      "I830.5" { ExternalVisible := 'False'} : Bool := FALSE;   // I830.5
      "I830.6" { ExternalVisible := 'False'} : Bool := FALSE;   // I830.6
      "I830.7" { ExternalVisible := 'False'} : Bool := FALSE;   // I830.7
      "I831.0" { ExternalVisible := 'False'} : Bool := FALSE;   // I831.0
      "I831.1" { ExternalVisible := 'False'} : Bool := FALSE;   // I831.1
      "I831.2" { ExternalVisible := 'False'} : Bool := FALSE;   // I831.2
      "I831.3" { ExternalVisible := 'False'} : Bool := FALSE;   // I831.3
      "I831.4" { ExternalVisible := 'False'} : Bool := FALSE;   // I831.4
      "I831.5" { ExternalVisible := 'False'} : Bool := FALSE;   // I831.5
      "I831.6" { ExternalVisible := 'False'} : Bool := FALSE;   // I831.6
      "I831.7" { ExternalVisible := 'False'} : Bool := FALSE;   // I831.7
      "I832.0" { ExternalVisible := 'False'} : Bool := FALSE;   // I832.0
      "I832.1" { ExternalVisible := 'False'} : Bool := FALSE;   // I832.1
      "I832.2" { ExternalVisible := 'False'} : Bool := FALSE;   // I832.2
      "I832.3" { ExternalVisible := 'False'} : Bool := FALSE;   // I832.3
      "I832.4" { ExternalVisible := 'False'} : Bool := FALSE;   // I832.4
      "I832.5" { ExternalVisible := 'False'} : Bool := FALSE;   // I832.5
      "I832.6" { ExternalVisible := 'False'} : Bool := FALSE;   // I832.6
      "I832.7" { ExternalVisible := 'False'} : Bool := FALSE;   // I832.7
      "I833.0" { ExternalVisible := 'False'} : Bool := FALSE;   // I833.0
      "I833.1" { ExternalVisible := 'False'} : Bool := FALSE;   // I833.1
      "I833.2" { ExternalVisible := 'False'} : Bool := FALSE;   // I833.2
      "I833.3" { ExternalVisible := 'False'} : Bool := FALSE;   // I833.3
      "I833.4" { ExternalVisible := 'False'} : Bool := FALSE;   // I833.4
      "I833.5" { ExternalVisible := 'False'} : Bool := FALSE;   // I833.5
      "I833.6" { ExternalVisible := 'False'} : Bool := FALSE;   // I833.6
      "I833.7" { ExternalVisible := 'False'} : Bool := FALSE;   // I833.7
      "I834.0" { ExternalVisible := 'False'} : Bool := FALSE;   // I834.0
      "I834.1" { ExternalVisible := 'False'} : Bool := FALSE;   // I834.1
      "I834.2" { ExternalVisible := 'False'} : Bool := FALSE;   // I834.2
      "I834.3" { ExternalVisible := 'False'} : Bool := FALSE;   // I834.3
      "I834.4" { ExternalVisible := 'False'} : Bool := FALSE;   // I834.4
      "I834.5" { ExternalVisible := 'False'} : Bool := FALSE;   // I834.5
      "I834.6" { ExternalVisible := 'False'} : Bool := FALSE;   // I834.6
      "I834.7" { ExternalVisible := 'False'} : Bool := FALSE;   // I834.7
      "I835.0" { ExternalVisible := 'False'} : Bool := FALSE;   // I835.0
      "I835.1" { ExternalVisible := 'False'} : Bool := FALSE;   // I835.1
      "I835.2" { ExternalVisible := 'False'} : Bool := FALSE;   // I835.2
      "I835.3" { ExternalVisible := 'False'} : Bool := FALSE;   // I835.3
      "I835.4" { ExternalVisible := 'False'} : Bool := FALSE;   // I835.4
      "I835.5" { ExternalVisible := 'False'} : Bool := FALSE;   // I835.5
      "I835.6" { ExternalVisible := 'False'} : Bool := FALSE;   // I835.6
      "I835.7" { ExternalVisible := 'False'} : Bool := FALSE;   // I835.7
      "I836.0" { ExternalVisible := 'False'} : Bool := FALSE;   // I836.0
      "I836.1" { ExternalVisible := 'False'} : Bool := FALSE;   // I836.1
      "I836.2" { ExternalVisible := 'False'} : Bool := FALSE;   // I836.2
      "I836.3" { ExternalVisible := 'False'} : Bool := FALSE;   // I836.3
      "I836.4" { ExternalVisible := 'False'} : Bool := FALSE;   // I836.4
      "I836.5" { ExternalVisible := 'False'} : Bool := FALSE;   // I836.5
      "I836.6" { ExternalVisible := 'False'} : Bool := FALSE;   // I836.6
      "I836.7" { ExternalVisible := 'False'} : Bool := FALSE;   // I836.7
      "I837.0" { ExternalVisible := 'False'} : Bool := FALSE;   // I837.0
      "I837.1" { ExternalVisible := 'False'} : Bool := FALSE;   // I837.1
      "I837.2" { ExternalVisible := 'False'} : Bool := FALSE;   // I837.2
      "I837.3" { ExternalVisible := 'False'} : Bool := FALSE;   // I837.3
      "I837.4" { ExternalVisible := 'False'} : Bool := FALSE;   // I837.4
      "I837.5" { ExternalVisible := 'False'} : Bool := FALSE;   // I837.5
      "I837.6" { ExternalVisible := 'False'} : Bool := FALSE;   // I837.6
      "I837.7" { ExternalVisible := 'False'} : Bool := FALSE;   // I837.7
      "I838.0" { ExternalVisible := 'False'} : Bool := FALSE;   // I838.0
      "I838.1" { ExternalVisible := 'False'} : Bool := FALSE;   // I838.1
      "I838.2" { ExternalVisible := 'False'} : Bool := FALSE;   // I838.2
      "I838.3" { ExternalVisible := 'False'} : Bool := FALSE;   // I838.3
      "I838.4" { ExternalVisible := 'False'} : Bool := FALSE;   // I838.4
      "I838.5" { ExternalVisible := 'False'} : Bool := FALSE;   // I838.5
      "I838.6" { ExternalVisible := 'False'} : Bool := FALSE;   // I838.6
      "I838.7" { ExternalVisible := 'False'} : Bool := FALSE;   // I838.7
      "I839.0" { ExternalVisible := 'False'} : Bool := FALSE;   // I839.0
      "I839.1" { ExternalVisible := 'False'} : Bool := FALSE;   // I839.1
      "I839.2" { ExternalVisible := 'False'} : Bool := FALSE;   // I839.2
      "I839.3" { ExternalVisible := 'False'} : Bool := FALSE;   // I839.3
      "I839.4" { ExternalVisible := 'False'} : Bool := FALSE;   // I839.4
      "I839.5" { ExternalVisible := 'False'} : Bool := FALSE;   // I839.5
      "I839.6" { ExternalVisible := 'False'} : Bool := FALSE;   // I839.6
      "I839.7" { ExternalVisible := 'False'} : Bool := FALSE;   // I839.7
      "I840.0" { ExternalVisible := 'False'} : Bool := FALSE;   // I840.0
      "I840.1" { ExternalVisible := 'False'} : Bool := FALSE;   // I840.1
      "I840.2" { ExternalVisible := 'False'} : Bool := FALSE;   // I840.2
      "I840.3" { ExternalVisible := 'False'} : Bool := FALSE;   // I840.3
      "I840.4" { ExternalVisible := 'False'} : Bool := FALSE;   // I840.4
      "I840.5" { ExternalVisible := 'False'} : Bool := FALSE;   // I840.5
      "I840.6" { ExternalVisible := 'False'} : Bool := FALSE;   // I840.6
      "I840.7" { ExternalVisible := 'False'} : Bool := FALSE;   // I840.7
      "I841.0" { ExternalVisible := 'False'} : Bool := FALSE;   // I841.0
      "I841.1" { ExternalVisible := 'False'} : Bool := FALSE;   // I841.1
      "I841.2" { ExternalVisible := 'False'} : Bool := FALSE;   // I841.2
      "I841.3" { ExternalVisible := 'False'} : Bool := FALSE;   // I841.3
      "I841.4" { ExternalVisible := 'False'} : Bool := FALSE;   // I841.4
      "I841.5" { ExternalVisible := 'False'} : Bool := FALSE;   // I841.5
      "I841.6" { ExternalVisible := 'False'} : Bool := FALSE;   // I841.6
      "I841.7" { ExternalVisible := 'False'} : Bool := FALSE;   // I841.7
      "I842.0" { ExternalVisible := 'False'} : Bool := FALSE;   // I842.0
      "I842.1" { ExternalVisible := 'False'} : Bool := FALSE;   // I842.1
      "I842.2" { ExternalVisible := 'False'} : Bool := FALSE;   // I842.2
      "I842.3" { ExternalVisible := 'False'} : Bool := FALSE;   // I842.3
      "I842.4" { ExternalVisible := 'False'} : Bool := FALSE;   // I842.4
      "I842.5" { ExternalVisible := 'False'} : Bool := FALSE;   // I842.5
      "I842.6" { ExternalVisible := 'False'} : Bool := FALSE;   // I842.6
      "I842.7" { ExternalVisible := 'False'} : Bool := FALSE;   // I842.7
      "I843.0" { ExternalVisible := 'False'} : Bool := FALSE;   // I843.0
      "I843.1" { ExternalVisible := 'False'} : Bool := FALSE;   // I843.1
      "I843.2" { ExternalVisible := 'False'} : Bool := FALSE;   // I843.2
      "I843.3" { ExternalVisible := 'False'} : Bool := FALSE;   // I843.3
      "I843.4" { ExternalVisible := 'False'} : Bool := FALSE;   // I843.4
      "I843.5" { ExternalVisible := 'False'} : Bool := FALSE;   // I843.5
      "I843.6" { ExternalVisible := 'False'} : Bool := FALSE;   // I843.6
      "I843.7" { ExternalVisible := 'False'} : Bool := FALSE;   // I843.7
      "I844.0" { ExternalVisible := 'False'} : Bool := FALSE;   // I844.0
      "I844.1" { ExternalVisible := 'False'} : Bool := FALSE;   // I844.1
      "I844.2" { ExternalVisible := 'False'} : Bool := FALSE;   // I844.2
      "I844.3" { ExternalVisible := 'False'} : Bool := FALSE;   // I844.3
      "I844.4" { ExternalVisible := 'False'} : Bool := FALSE;   // I844.4
      "I844.5" { ExternalVisible := 'False'} : Bool := FALSE;   // I844.5
      "I844.6" { ExternalVisible := 'False'} : Bool := FALSE;   // I844.6
      "I844.7" { ExternalVisible := 'False'} : Bool := FALSE;   // I844.7
      "I845.0" { ExternalVisible := 'False'} : Bool := FALSE;   // I845.0
      "I845.1" { ExternalVisible := 'False'} : Bool := FALSE;   // I845.1
      "I845.2" { ExternalVisible := 'False'} : Bool := FALSE;   // I845.2
      "I845.3" { ExternalVisible := 'False'} : Bool := FALSE;   // I845.3
      "I845.4" { ExternalVisible := 'False'} : Bool := FALSE;   // I845.4
      "I845.5" { ExternalVisible := 'False'} : Bool := FALSE;   // I845.5
      "I845.6" { ExternalVisible := 'False'} : Bool := FALSE;   // I845.6
      "I845.7" { ExternalVisible := 'False'} : Bool := FALSE;   // I845.7
      "I846.0" { ExternalVisible := 'False'} : Bool := FALSE;   // I846.0
      "I846.1" { ExternalVisible := 'False'} : Bool := FALSE;   // I846.1
      "I846.2" { ExternalVisible := 'False'} : Bool := FALSE;   // I846.2
      "I846.3" { ExternalVisible := 'False'} : Bool := FALSE;   // I846.3
      "I846.4" { ExternalVisible := 'False'} : Bool := FALSE;   // I846.4
      "I846.5" { ExternalVisible := 'False'} : Bool := FALSE;   // I846.5
      "I846.6" { ExternalVisible := 'False'} : Bool := FALSE;   // I846.6
      "I846.7" { ExternalVisible := 'False'} : Bool := FALSE;   // I846.7
      "I847.0" { ExternalVisible := 'False'} : Bool := FALSE;   // I847.0
      "I847.1" { ExternalVisible := 'False'} : Bool := FALSE;   // I847.1
      "I847.2" { ExternalVisible := 'False'} : Bool := FALSE;   // I847.2
      "I847.3" { ExternalVisible := 'False'} : Bool := FALSE;   // I847.3
      "I847.4" { ExternalVisible := 'False'} : Bool := FALSE;   // I847.4
      "I847.5" { ExternalVisible := 'False'} : Bool := FALSE;   // I847.5
      "I847.6" { ExternalVisible := 'False'} : Bool := FALSE;   // I847.6
      "I847.7" { ExternalVisible := 'False'} : Bool := FALSE;   // I847.7
      "I848.0" { ExternalVisible := 'False'} : Bool := FALSE;   // I848.0
      "I848.1" { ExternalVisible := 'False'} : Bool := FALSE;   // I848.1
      "I848.2" { ExternalVisible := 'False'} : Bool := FALSE;   // I848.2
      "I848.3" { ExternalVisible := 'False'} : Bool := FALSE;   // I848.3
      "I848.4" { ExternalVisible := 'False'} : Bool := FALSE;   // I848.4
      "I848.5" { ExternalVisible := 'False'} : Bool := FALSE;   // I848.5
      "I848.6" { ExternalVisible := 'False'} : Bool := FALSE;   // I848.6
      "I848.7" { ExternalVisible := 'False'} : Bool := FALSE;   // I848.7
      "I849.0" { ExternalVisible := 'False'} : Bool := FALSE;   // I849.0
      "I849.1" { ExternalVisible := 'False'} : Bool := FALSE;   // I849.1
      "I849.2" { ExternalVisible := 'False'} : Bool := FALSE;   // I849.2
      "I849.3" { ExternalVisible := 'False'} : Bool := FALSE;   // I849.3
      "I849.4" { ExternalVisible := 'False'} : Bool := FALSE;   // I849.4
      "I849.5" { ExternalVisible := 'False'} : Bool := FALSE;   // I849.5
      "I849.6" { ExternalVisible := 'False'} : Bool := FALSE;   // I849.6
      "I849.7" { ExternalVisible := 'False'} : Bool := FALSE;   // I849.7
      "I850.0" { ExternalVisible := 'False'} : Bool := FALSE;   // I850.0
      "I850.1" { ExternalVisible := 'False'} : Bool := FALSE;   // I850.1
      "I850.2" { ExternalVisible := 'False'} : Bool := FALSE;   // I850.2
      "I850.3" { ExternalVisible := 'False'} : Bool := FALSE;   // I850.3
      "I850.4" { ExternalVisible := 'False'} : Bool := FALSE;   // I850.4
      "I850.5" { ExternalVisible := 'False'} : Bool := FALSE;   // I850.5
      "I850.6" { ExternalVisible := 'False'} : Bool := FALSE;   // I850.6
      "I850.7" { ExternalVisible := 'False'} : Bool := FALSE;   // I850.7
      "I851.0" { ExternalVisible := 'False'} : Bool := FALSE;   // I851.0
      "I851.1" { ExternalVisible := 'False'} : Bool := FALSE;   // I851.1
      "I851.2" { ExternalVisible := 'False'} : Bool := FALSE;   // I851.2
      "I851.3" { ExternalVisible := 'False'} : Bool := FALSE;   // I851.3
      "I851.4" { ExternalVisible := 'False'} : Bool := FALSE;   // I851.4
      "I851.5" { ExternalVisible := 'False'} : Bool := FALSE;   // I851.5
      "I851.6" { ExternalVisible := 'False'} : Bool := FALSE;   // I851.6
      "I851.7" { ExternalVisible := 'False'} : Bool := FALSE;   // I851.7
      "I852.0" { ExternalVisible := 'False'} : Bool := FALSE;   // I852.0
      "I852.1" { ExternalVisible := 'False'} : Bool := FALSE;   // I852.1
      "I852.2" { ExternalVisible := 'False'} : Bool := FALSE;   // I852.2
      "I852.3" { ExternalVisible := 'False'} : Bool := FALSE;   // I852.3
      "I852.4" { ExternalVisible := 'False'} : Bool := FALSE;   // I852.4
      "I852.5" { ExternalVisible := 'False'} : Bool := FALSE;   // I852.5
      "I852.6" { ExternalVisible := 'False'} : Bool := FALSE;   // I852.6
      "I852.7" { ExternalVisible := 'False'} : Bool := FALSE;   // I852.7
      "I853.0" { ExternalVisible := 'False'} : Bool := FALSE;   // I853.0
      "I853.1" { ExternalVisible := 'False'} : Bool := FALSE;   // I853.1
      "I853.2" { ExternalVisible := 'False'} : Bool := FALSE;   // I853.2
      "I853.3" { ExternalVisible := 'False'} : Bool := FALSE;   // I853.3
      "I853.4" { ExternalVisible := 'False'} : Bool := FALSE;   // I853.4
      "I853.5" { ExternalVisible := 'False'} : Bool := FALSE;   // I853.5
      "I853.6" { ExternalVisible := 'False'} : Bool := FALSE;   // I853.6
      "I853.7" { ExternalVisible := 'False'} : Bool := FALSE;   // I853.7
      "I854.0" { ExternalVisible := 'False'} : Bool := FALSE;   // I854.0
      "I854.1" { ExternalVisible := 'False'} : Bool := FALSE;   // I854.1
      "I854.2" { ExternalVisible := 'False'} : Bool := FALSE;   // I854.2
      "I854.3" { ExternalVisible := 'False'} : Bool := FALSE;   // I854.3
      "I854.4" { ExternalVisible := 'False'} : Bool := FALSE;   // I854.4
      "I854.5" { ExternalVisible := 'False'} : Bool := FALSE;   // I854.5
      "I854.6" { ExternalVisible := 'False'} : Bool := FALSE;   // I854.6
      "I854.7" { ExternalVisible := 'False'} : Bool := FALSE;   // I854.7
      "I855.0" { ExternalVisible := 'False'} : Bool := FALSE;   // I855.0
      "I855.1" { ExternalVisible := 'False'} : Bool := FALSE;   // I855.1
      "I855.2" { ExternalVisible := 'False'} : Bool := FALSE;   // I855.2
      "I855.3" { ExternalVisible := 'False'} : Bool := FALSE;   // I855.3
      "I855.4" { ExternalVisible := 'False'} : Bool := FALSE;   // I855.4
      "I855.5" { ExternalVisible := 'False'} : Bool := FALSE;   // I855.5
      "I855.6" { ExternalVisible := 'False'} : Bool := FALSE;   // I855.6
      "I855.7" { ExternalVisible := 'False'} : Bool := FALSE;   // I855.7
      "I856.0" { ExternalVisible := 'False'} : Bool := FALSE;   // I856.0
      "I856.1" { ExternalVisible := 'False'} : Bool := FALSE;   // I856.1
      "I856.2" { ExternalVisible := 'False'} : Bool := FALSE;   // I856.2
      "I856.3" { ExternalVisible := 'False'} : Bool := FALSE;   // I856.3
      "I856.4" { ExternalVisible := 'False'} : Bool := FALSE;   // I856.4
      "I856.5" { ExternalVisible := 'False'} : Bool := FALSE;   // I856.5
      "I856.6" { ExternalVisible := 'False'} : Bool := FALSE;   // I856.6
      "I856.7" { ExternalVisible := 'False'} : Bool := FALSE;   // I856.7
      "I857.0" { ExternalVisible := 'False'} : Bool := FALSE;   // I857.0
      "I857.1" { ExternalVisible := 'False'} : Bool := FALSE;   // I857.1
      "I857.2" { ExternalVisible := 'False'} : Bool := FALSE;   // I857.2
      "I857.3" { ExternalVisible := 'False'} : Bool := FALSE;   // I857.3
      "I857.4" { ExternalVisible := 'False'} : Bool := FALSE;   // I857.4
      "I857.5" { ExternalVisible := 'False'} : Bool := FALSE;   // I857.5
      "I857.6" { ExternalVisible := 'False'} : Bool := FALSE;   // I857.6
      "I857.7" { ExternalVisible := 'False'} : Bool := FALSE;   // I857.7
      "I858.0" { ExternalVisible := 'False'} : Bool := FALSE;   // I858.0
      "I858.1" { ExternalVisible := 'False'} : Bool := FALSE;   // I858.1
      "I858.2" { ExternalVisible := 'False'} : Bool := FALSE;   // I858.2
      "I858.3" { ExternalVisible := 'False'} : Bool := FALSE;   // I858.3
      "I858.4" { ExternalVisible := 'False'} : Bool := FALSE;   // I858.4
      "I858.5" { ExternalVisible := 'False'} : Bool := FALSE;   // I858.5
      "I858.6" { ExternalVisible := 'False'} : Bool := FALSE;   // I858.6
      "I858.7" { ExternalVisible := 'False'} : Bool := FALSE;   // I858.7
      "I859.0" { ExternalVisible := 'False'} : Bool := FALSE;   // I859.0
      "I859.1" { ExternalVisible := 'False'} : Bool := FALSE;   // I859.1
      "I859.2" { ExternalVisible := 'False'} : Bool := FALSE;   // I859.2
      "I859.3" { ExternalVisible := 'False'} : Bool := FALSE;   // I859.3
      "I859.4" { ExternalVisible := 'False'} : Bool := FALSE;   // I859.4
      "I859.5" { ExternalVisible := 'False'} : Bool := FALSE;   // I859.5
      "I859.6" { ExternalVisible := 'False'} : Bool := FALSE;   // I859.6
      "I859.7" { ExternalVisible := 'False'} : Bool := FALSE;   // I859.7
      "I860.0" { ExternalVisible := 'False'} : Bool := FALSE;   // I860.0
      "I860.1" { ExternalVisible := 'False'} : Bool := FALSE;   // I860.1
      "I860.2" { ExternalVisible := 'False'} : Bool := FALSE;   // I860.2
      "I860.3" { ExternalVisible := 'False'} : Bool := FALSE;   // I860.3
      "I860.4" { ExternalVisible := 'False'} : Bool := FALSE;   // I860.4
      "I860.5" { ExternalVisible := 'False'} : Bool := FALSE;   // I860.5
      "I860.6" { ExternalVisible := 'False'} : Bool := FALSE;   // I860.6
      "I860.7" { ExternalVisible := 'False'} : Bool := FALSE;   // I860.7
      "I861.0" { ExternalVisible := 'False'} : Bool := FALSE;   // I861.0
      "I861.1" { ExternalVisible := 'False'} : Bool := FALSE;   // I861.1
      "I861.2" { ExternalVisible := 'False'} : Bool := FALSE;   // I861.2
      "I861.3" { ExternalVisible := 'False'} : Bool := FALSE;   // I861.3
      "I861.4" { ExternalVisible := 'False'} : Bool := FALSE;   // I861.4
      "I861.5" { ExternalVisible := 'False'} : Bool := FALSE;   // I861.5
      "I861.6" { ExternalVisible := 'False'} : Bool := FALSE;   // I861.6
      "I861.7" { ExternalVisible := 'False'} : Bool := FALSE;   // I861.7
      "I862.0" { ExternalVisible := 'False'} : Bool := FALSE;   // I862.0
      "I862.1" { ExternalVisible := 'False'} : Bool := FALSE;   // I862.1
      "I862.2" { ExternalVisible := 'False'} : Bool := FALSE;   // I862.2
      "I862.3" { ExternalVisible := 'False'} : Bool := FALSE;   // I862.3
      "I862.4" { ExternalVisible := 'False'} : Bool := FALSE;   // I862.4
      "I862.5" { ExternalVisible := 'False'} : Bool := FALSE;   // I862.5
      "I862.6" { ExternalVisible := 'False'} : Bool := FALSE;   // I862.6
      "I862.7" { ExternalVisible := 'False'} : Bool := FALSE;   // I862.7
      "I863.0" { ExternalVisible := 'False'} : Bool := FALSE;   // I863.0
      "I863.1" { ExternalVisible := 'False'} : Bool := FALSE;   // I863.1
      "I863.2" { ExternalVisible := 'False'} : Bool := FALSE;   // I863.2
      "I863.3" { ExternalVisible := 'False'} : Bool := FALSE;   // I863.3
      "I863.4" { ExternalVisible := 'False'} : Bool := FALSE;   // I863.4
      "I863.5" { ExternalVisible := 'False'} : Bool := FALSE;   // I863.5
      "I863.6" { ExternalVisible := 'False'} : Bool := FALSE;   // I863.6
      "I863.7" { ExternalVisible := 'False'} : Bool := FALSE;   // I863.7
      "I864.0" { ExternalVisible := 'False'} : Bool := FALSE;   // I864.0
      "I864.1" { ExternalVisible := 'False'} : Bool := FALSE;   // I864.1
      "I864.2" { ExternalVisible := 'False'} : Bool := FALSE;   // I864.2
      "I864.3" { ExternalVisible := 'False'} : Bool := FALSE;   // I864.3
      "I864.4" { ExternalVisible := 'False'} : Bool := FALSE;   // I864.4
      "I864.5" { ExternalVisible := 'False'} : Bool := FALSE;   // I864.5
      "I864.6" { ExternalVisible := 'False'} : Bool := FALSE;   // I864.6
      "I864.7" { ExternalVisible := 'False'} : Bool := FALSE;   // I864.7
      "I865.0" { ExternalVisible := 'False'} : Bool := FALSE;   // I865.0
      "I865.1" { ExternalVisible := 'False'} : Bool := FALSE;   // I865.1
      "I865.2" { ExternalVisible := 'False'} : Bool := FALSE;   // I865.2
      "I865.3" { ExternalVisible := 'False'} : Bool := FALSE;   // I865.3
      "I865.4" { ExternalVisible := 'False'} : Bool := FALSE;   // I865.4
      "I865.5" { ExternalVisible := 'False'} : Bool := FALSE;   // I865.5
      "I865.6" { ExternalVisible := 'False'} : Bool := FALSE;   // I865.6
      "I865.7" { ExternalVisible := 'False'} : Bool := FALSE;   // I865.7
      "I866.0" { ExternalVisible := 'False'} : Bool := FALSE;   // I866.0
      "I866.1" { ExternalVisible := 'False'} : Bool := FALSE;   // I866.1
      "I866.2" { ExternalVisible := 'False'} : Bool := FALSE;   // I866.2
      "I866.3" { ExternalVisible := 'False'} : Bool := FALSE;   // I866.3
      "I866.4" { ExternalVisible := 'False'} : Bool := FALSE;   // I866.4
      "I866.5" { ExternalVisible := 'False'} : Bool := FALSE;   // I866.5
      "I866.6" { ExternalVisible := 'False'} : Bool := FALSE;   // I866.6
      "I866.7" { ExternalVisible := 'False'} : Bool := FALSE;   // I866.7
      "I867.0" { ExternalVisible := 'False'} : Bool := FALSE;   // I867.0
      "I867.1" { ExternalVisible := 'False'} : Bool := FALSE;   // I867.1
      "I867.2" { ExternalVisible := 'False'} : Bool := FALSE;   // I867.2
      "I867.3" { ExternalVisible := 'False'} : Bool := FALSE;   // I867.3
      "I867.4" { ExternalVisible := 'False'} : Bool := FALSE;   // I867.4
      "I867.5" { ExternalVisible := 'False'} : Bool := FALSE;   // I867.5
      "I867.6" { ExternalVisible := 'False'} : Bool := FALSE;   // I867.6
      "I867.7" { ExternalVisible := 'False'} : Bool := FALSE;   // I867.7
      "I868.0" { ExternalVisible := 'False'} : Bool := FALSE;   // I868.0
      "I868.1" { ExternalVisible := 'False'} : Bool := FALSE;   // I868.1
      "I868.2" { ExternalVisible := 'False'} : Bool := FALSE;   // I868.2
      "I868.3" { ExternalVisible := 'False'} : Bool := FALSE;   // I868.3
      "I868.4" { ExternalVisible := 'False'} : Bool := FALSE;   // I868.4
      "I868.5" { ExternalVisible := 'False'} : Bool := FALSE;   // I868.5
      "I868.6" { ExternalVisible := 'False'} : Bool := FALSE;   // I868.6
      "I868.7" { ExternalVisible := 'False'} : Bool := FALSE;   // I868.7
      "I869.0" { ExternalVisible := 'False'} : Bool := FALSE;   // I869.0
      "I869.1" { ExternalVisible := 'False'} : Bool := FALSE;   // I869.1
      "I869.2" { ExternalVisible := 'False'} : Bool := FALSE;   // I869.2
      "I869.3" { ExternalVisible := 'False'} : Bool := FALSE;   // I869.3
      "I869.4" { ExternalVisible := 'False'} : Bool := FALSE;   // I869.4
      "I869.5" { ExternalVisible := 'False'} : Bool := FALSE;   // I869.5
      "I869.6" { ExternalVisible := 'False'} : Bool := FALSE;   // I869.6
      "I869.7" { ExternalVisible := 'False'} : Bool := FALSE;   // I869.7
      "I870.0" { ExternalVisible := 'False'} : Bool := FALSE;   // I870.0
      "I870.1" { ExternalVisible := 'False'} : Bool := FALSE;   // I870.1
      "I870.2" { ExternalVisible := 'False'} : Bool := FALSE;   // I870.2
      "I870.3" { ExternalVisible := 'False'} : Bool := FALSE;   // I870.3
      "I870.4" { ExternalVisible := 'False'} : Bool := FALSE;   // I870.4
      "I870.5" { ExternalVisible := 'False'} : Bool := FALSE;   // I870.5
      "I870.6" { ExternalVisible := 'False'} : Bool := FALSE;   // I870.6
      "I870.7" { ExternalVisible := 'False'} : Bool := FALSE;   // I870.7
      "I871.0" { ExternalVisible := 'False'} : Bool := FALSE;   // I871.0
      "I871.1" { ExternalVisible := 'False'} : Bool := FALSE;   // I871.1
      "I871.2" { ExternalVisible := 'False'} : Bool := FALSE;   // I871.2
      "I871.3" { ExternalVisible := 'False'} : Bool := FALSE;   // I871.3
      "I871.4" { ExternalVisible := 'False'} : Bool := FALSE;   // I871.4
      "I871.5" { ExternalVisible := 'False'} : Bool := FALSE;   // I871.5
      "I871.6" { ExternalVisible := 'False'} : Bool := FALSE;   // I871.6
      "I871.7" { ExternalVisible := 'False'} : Bool := FALSE;   // I871.7
      "I872.0" { ExternalVisible := 'False'} : Bool := FALSE;   // I872.0
      "I872.1" { ExternalVisible := 'False'} : Bool := FALSE;   // I872.1
      "I872.2" { ExternalVisible := 'False'} : Bool := FALSE;   // I872.2
      "I872.3" { ExternalVisible := 'False'} : Bool := FALSE;   // I872.3
      "I872.4" { ExternalVisible := 'False'} : Bool := FALSE;   // I872.4
      "I872.5" { ExternalVisible := 'False'} : Bool := FALSE;   // I872.5
      "I872.6" { ExternalVisible := 'False'} : Bool := FALSE;   // I872.6
      "I872.7" { ExternalVisible := 'False'} : Bool := FALSE;   // I872.7
      "I873.0" { ExternalVisible := 'False'} : Bool := FALSE;   // I873.0
      "I873.1" { ExternalVisible := 'False'} : Bool := FALSE;   // I873.1
      "I873.2" { ExternalVisible := 'False'} : Bool := FALSE;   // I873.2
      "I873.3" { ExternalVisible := 'False'} : Bool := FALSE;   // I873.3
      "I873.4" { ExternalVisible := 'False'} : Bool := FALSE;   // I873.4
      "I873.5" { ExternalVisible := 'False'} : Bool := FALSE;   // I873.5
      "I873.6" { ExternalVisible := 'False'} : Bool := FALSE;   // I873.6
      "I873.7" { ExternalVisible := 'False'} : Bool := FALSE;   // I873.7
      "I874.0" { ExternalVisible := 'False'} : Bool := FALSE;   // I874.0
      "I874.1" { ExternalVisible := 'False'} : Bool := FALSE;   // I874.1
      "I874.2" { ExternalVisible := 'False'} : Bool := FALSE;   // I874.2
      "I874.3" { ExternalVisible := 'False'} : Bool := FALSE;   // I874.3
      "I874.4" { ExternalVisible := 'False'} : Bool := FALSE;   // I874.4
      "I874.5" { ExternalVisible := 'False'} : Bool := FALSE;   // I874.5
      "I874.6" { ExternalVisible := 'False'} : Bool := FALSE;   // I874.6
      "I874.7" { ExternalVisible := 'False'} : Bool := FALSE;   // I874.7
      "I875.0" { ExternalVisible := 'False'} : Bool := FALSE;   // I875.0
      "I875.1" { ExternalVisible := 'False'} : Bool := FALSE;   // I875.1
      "I875.2" { ExternalVisible := 'False'} : Bool := FALSE;   // I875.2
      "I875.3" { ExternalVisible := 'False'} : Bool := FALSE;   // I875.3
      "I875.4" { ExternalVisible := 'False'} : Bool := FALSE;   // I875.4
      "I875.5" { ExternalVisible := 'False'} : Bool := FALSE;   // I875.5
      "I875.6" { ExternalVisible := 'False'} : Bool := FALSE;   // I875.6
      "I875.7" { ExternalVisible := 'False'} : Bool := FALSE;   // I875.7
      "I876.0" { ExternalVisible := 'False'} : Bool := FALSE;   // I876.0
      "I876.1" { ExternalVisible := 'False'} : Bool := FALSE;   // I876.1
      "I876.2" { ExternalVisible := 'False'} : Bool := FALSE;   // I876.2
      "I876.3" { ExternalVisible := 'False'} : Bool := FALSE;   // I876.3
      "I876.4" { ExternalVisible := 'False'} : Bool := FALSE;   // I876.4
      "I876.5" { ExternalVisible := 'False'} : Bool := FALSE;   // I876.5
      "I876.6" { ExternalVisible := 'False'} : Bool := FALSE;   // I876.6
      "I876.7" { ExternalVisible := 'False'} : Bool := FALSE;   // I876.7
      "I877.0" { ExternalVisible := 'False'} : Bool := FALSE;   // I877.0
      "I877.1" { ExternalVisible := 'False'} : Bool := FALSE;   // I877.1
      "I877.2" { ExternalVisible := 'False'} : Bool := FALSE;   // I877.2
      "I877.3" { ExternalVisible := 'False'} : Bool := FALSE;   // I877.3
      "I877.4" { ExternalVisible := 'False'} : Bool := FALSE;   // I877.4
      "I877.5" { ExternalVisible := 'False'} : Bool := FALSE;   // I877.5
      "I877.6" { ExternalVisible := 'False'} : Bool := FALSE;   // I877.6
      "I877.7" { ExternalVisible := 'False'} : Bool := FALSE;   // I877.7
      "I878.0" { ExternalVisible := 'False'} : Bool := FALSE;   // I878.0
      "I878.1" { ExternalVisible := 'False'} : Bool := FALSE;   // I878.1
      "I878.2" { ExternalVisible := 'False'} : Bool := FALSE;   // I878.2
      "I878.3" { ExternalVisible := 'False'} : Bool := FALSE;   // I878.3
      "I878.4" { ExternalVisible := 'False'} : Bool := FALSE;   // I878.4
      "I878.5" { ExternalVisible := 'False'} : Bool := FALSE;   // I878.5
      "I878.6" { ExternalVisible := 'False'} : Bool := FALSE;   // I878.6
      "I878.7" { ExternalVisible := 'False'} : Bool := FALSE;   // I878.7
      "I879.0" { ExternalVisible := 'False'} : Bool := FALSE;   // I879.0
      "I879.1" { ExternalVisible := 'False'} : Bool := FALSE;   // I879.1
      "I879.2" { ExternalVisible := 'False'} : Bool := FALSE;   // I879.2
      "I879.3" { ExternalVisible := 'False'} : Bool := FALSE;   // I879.3
      "I879.4" { ExternalVisible := 'False'} : Bool := FALSE;   // I879.4
      "I879.5" { ExternalVisible := 'False'} : Bool := FALSE;   // I879.5
      "I879.6" { ExternalVisible := 'False'} : Bool := FALSE;   // I879.6
      "I879.7" { ExternalVisible := 'False'} : Bool := FALSE;   // I879.7
      "I880.0" { ExternalVisible := 'False'} : Bool := FALSE;   // I880.0
      "I880.1" { ExternalVisible := 'False'} : Bool := FALSE;   // I880.1
      "I880.2" { ExternalVisible := 'False'} : Bool := FALSE;   // I880.2
      "I880.3" { ExternalVisible := 'False'} : Bool := FALSE;   // I880.3
      "I880.4" { ExternalVisible := 'False'} : Bool := FALSE;   // I880.4
      "I880.5" { ExternalVisible := 'False'} : Bool := FALSE;   // I880.5
      "I880.6" { ExternalVisible := 'False'} : Bool := FALSE;   // I880.6
      "I880.7" { ExternalVisible := 'False'} : Bool := FALSE;   // I880.7
      "I881.0" { ExternalVisible := 'False'} : Bool := FALSE;   // I881.0
      "I881.1" { ExternalVisible := 'False'} : Bool := FALSE;   // I881.1
      "I881.2" { ExternalVisible := 'False'} : Bool := FALSE;   // I881.2
      "I881.3" { ExternalVisible := 'False'} : Bool := FALSE;   // I881.3
      "I881.4" { ExternalVisible := 'False'} : Bool := FALSE;   // I881.4
      "I881.5" { ExternalVisible := 'False'} : Bool := FALSE;   // I881.5
      "I881.6" { ExternalVisible := 'False'} : Bool := FALSE;   // I881.6
      "I881.7" { ExternalVisible := 'False'} : Bool := FALSE;   // I881.7
      "I882.0" { ExternalVisible := 'False'} : Bool := FALSE;   // I882.0
      "I882.1" { ExternalVisible := 'False'} : Bool := FALSE;   // I882.1
      "I882.2" { ExternalVisible := 'False'} : Bool := FALSE;   // I882.2
      "I882.3" { ExternalVisible := 'False'} : Bool := FALSE;   // I882.3
      "I882.4" { ExternalVisible := 'False'} : Bool := FALSE;   // I882.4
      "I882.5" { ExternalVisible := 'False'} : Bool := FALSE;   // I882.5
      "I882.6" { ExternalVisible := 'False'} : Bool := FALSE;   // I882.6
      "I882.7" { ExternalVisible := 'False'} : Bool := FALSE;   // I882.7
      "I883.0" { ExternalVisible := 'False'} : Bool := FALSE;   // I883.0
      "I883.1" { ExternalVisible := 'False'} : Bool := FALSE;   // I883.1
      "I883.2" { ExternalVisible := 'False'} : Bool := FALSE;   // I883.2
      "I883.3" { ExternalVisible := 'False'} : Bool := FALSE;   // I883.3
      "I883.4" { ExternalVisible := 'False'} : Bool := FALSE;   // I883.4
      "I883.5" { ExternalVisible := 'False'} : Bool := FALSE;   // I883.5
      "I883.6" { ExternalVisible := 'False'} : Bool := FALSE;   // I883.6
      "I883.7" { ExternalVisible := 'False'} : Bool := FALSE;   // I883.7
      "I884.0" { ExternalVisible := 'False'} : Bool := FALSE;   // I884.0
      "I884.1" { ExternalVisible := 'False'} : Bool := FALSE;   // I884.1
      "I884.2" { ExternalVisible := 'False'} : Bool := FALSE;   // I884.2
      "I884.3" { ExternalVisible := 'False'} : Bool := FALSE;   // I884.3
      "I884.4" { ExternalVisible := 'False'} : Bool := FALSE;   // I884.4
      "I884.5" { ExternalVisible := 'False'} : Bool := FALSE;   // I884.5
      "I884.6" { ExternalVisible := 'False'} : Bool := FALSE;   // I884.6
      "I884.7" { ExternalVisible := 'False'} : Bool := FALSE;   // I884.7
      "I885.0" { ExternalVisible := 'False'} : Bool := FALSE;   // I885.0
      "I885.1" { ExternalVisible := 'False'} : Bool := FALSE;   // I885.1
      "I885.2" { ExternalVisible := 'False'} : Bool := FALSE;   // I885.2
      "I885.3" { ExternalVisible := 'False'} : Bool := FALSE;   // I885.3
      "I885.4" { ExternalVisible := 'False'} : Bool := FALSE;   // I885.4
      "I885.5" { ExternalVisible := 'False'} : Bool := FALSE;   // I885.5
      "I885.6" { ExternalVisible := 'False'} : Bool := FALSE;   // I885.6
      "I885.7" { ExternalVisible := 'False'} : Bool := FALSE;   // I885.7
      "I886.0" { ExternalVisible := 'False'} : Bool := FALSE;   // I886.0
      "I886.1" { ExternalVisible := 'False'} : Bool := FALSE;   // I886.1
      "I886.2" { ExternalVisible := 'False'} : Bool := FALSE;   // I886.2
      "I886.3" { ExternalVisible := 'False'} : Bool := FALSE;   // I886.3
      "I886.4" { ExternalVisible := 'False'} : Bool := FALSE;   // I886.4
      "I886.5" { ExternalVisible := 'False'} : Bool := FALSE;   // I886.5
      "I886.6" { ExternalVisible := 'False'} : Bool := FALSE;   // I886.6
      "I886.7" { ExternalVisible := 'False'} : Bool := FALSE;   // I886.7
      "I887.0" { ExternalVisible := 'False'} : Bool := FALSE;   // I887.0
      "I887.1" { ExternalVisible := 'False'} : Bool := FALSE;   // I887.1
      "I887.2" { ExternalVisible := 'False'} : Bool := FALSE;   // I887.2
      "I887.3" { ExternalVisible := 'False'} : Bool := FALSE;   // I887.3
      "I887.4" { ExternalVisible := 'False'} : Bool := FALSE;   // I887.4
      "I887.5" { ExternalVisible := 'False'} : Bool := FALSE;   // I887.5
      "I887.6" { ExternalVisible := 'False'} : Bool := FALSE;   // I887.6
      "I887.7" { ExternalVisible := 'False'} : Bool := FALSE;   // I887.7
      "I888.0" { ExternalVisible := 'False'} : Bool := FALSE;   // I888.0
      "I888.1" { ExternalVisible := 'False'} : Bool := FALSE;   // I888.1
      "I888.2" { ExternalVisible := 'False'} : Bool := FALSE;   // I888.2
      "I888.3" { ExternalVisible := 'False'} : Bool := FALSE;   // I888.3
      "I888.4" { ExternalVisible := 'False'} : Bool := FALSE;   // I888.4
      "I888.5" { ExternalVisible := 'False'} : Bool := FALSE;   // I888.5
      "I888.6" { ExternalVisible := 'False'} : Bool := FALSE;   // I888.6
      "I888.7" { ExternalVisible := 'False'} : Bool := FALSE;   // I888.7
      "I889.0" { ExternalVisible := 'False'} : Bool := FALSE;   // I889.0
      "I889.1" { ExternalVisible := 'False'} : Bool := FALSE;   // I889.1
      "I889.2" { ExternalVisible := 'False'} : Bool := FALSE;   // I889.2
      "I889.3" { ExternalVisible := 'False'} : Bool := FALSE;   // I889.3
      "I889.4" { ExternalVisible := 'False'} : Bool := FALSE;   // I889.4
      "I889.5" { ExternalVisible := 'False'} : Bool := FALSE;   // I889.5
      "I889.6" { ExternalVisible := 'False'} : Bool := FALSE;   // I889.6
      "I889.7" { ExternalVisible := 'False'} : Bool := FALSE;   // I889.7
      "I890.0" { ExternalVisible := 'False'} : Bool := FALSE;   // I890.0
      "I890.1" { ExternalVisible := 'False'} : Bool := FALSE;   // I890.1
      "I890.2" { ExternalVisible := 'False'} : Bool := FALSE;   // I890.2
      "I890.3" { ExternalVisible := 'False'} : Bool := FALSE;   // I890.3
      "I890.4" { ExternalVisible := 'False'} : Bool := FALSE;   // I890.4
      "I890.5" { ExternalVisible := 'False'} : Bool := FALSE;   // I890.5
      "I890.6" { ExternalVisible := 'False'} : Bool := FALSE;   // I890.6
      "I890.7" { ExternalVisible := 'False'} : Bool := FALSE;   // I890.7
      "I891.0" { ExternalVisible := 'False'} : Bool := FALSE;   // I891.0
      "I891.1" { ExternalVisible := 'False'} : Bool := FALSE;   // I891.1
      "I891.2" { ExternalVisible := 'False'} : Bool := FALSE;   // I891.2
      "I891.3" { ExternalVisible := 'False'} : Bool := FALSE;   // I891.3
      "I891.4" { ExternalVisible := 'False'} : Bool := FALSE;   // I891.4
      "I891.5" { ExternalVisible := 'False'} : Bool := FALSE;   // I891.5
      "I891.6" { ExternalVisible := 'False'} : Bool := FALSE;   // I891.6
      "I891.7" { ExternalVisible := 'False'} : Bool := FALSE;   // I891.7
      "I892.0" { ExternalVisible := 'False'} : Bool := FALSE;   // I892.0
      "I892.1" { ExternalVisible := 'False'} : Bool := FALSE;   // I892.1
      "I892.2" { ExternalVisible := 'False'} : Bool := FALSE;   // I892.2
      "I892.3" { ExternalVisible := 'False'} : Bool := FALSE;   // I892.3
      "I892.4" { ExternalVisible := 'False'} : Bool := FALSE;   // I892.4
      "I892.5" { ExternalVisible := 'False'} : Bool := FALSE;   // I892.5
      "I892.6" { ExternalVisible := 'False'} : Bool := FALSE;   // I892.6
      "I892.7" { ExternalVisible := 'False'} : Bool := FALSE;   // I892.7
      "I893.0" { ExternalVisible := 'False'} : Bool := FALSE;   // I893.0
      "I893.1" { ExternalVisible := 'False'} : Bool := FALSE;   // I893.1
      "I893.2" { ExternalVisible := 'False'} : Bool := FALSE;   // I893.2
      "I893.3" { ExternalVisible := 'False'} : Bool := FALSE;   // I893.3
      "I893.4" { ExternalVisible := 'False'} : Bool := FALSE;   // I893.4
      "I893.5" { ExternalVisible := 'False'} : Bool := FALSE;   // I893.5
      "I893.6" { ExternalVisible := 'False'} : Bool := FALSE;   // I893.6
      "I893.7" { ExternalVisible := 'False'} : Bool := FALSE;   // I893.7
      "I894.0" { ExternalVisible := 'False'} : Bool := FALSE;   // I894.0
      "I894.1" { ExternalVisible := 'False'} : Bool := FALSE;   // I894.1
      "I894.2" { ExternalVisible := 'False'} : Bool := FALSE;   // I894.2
      "I894.3" { ExternalVisible := 'False'} : Bool := FALSE;   // I894.3
      "I894.4" { ExternalVisible := 'False'} : Bool := FALSE;   // I894.4
      "I894.5" { ExternalVisible := 'False'} : Bool := FALSE;   // I894.5
      "I894.6" { ExternalVisible := 'False'} : Bool := FALSE;   // I894.6
      "I894.7" { ExternalVisible := 'False'} : Bool := FALSE;   // I894.7
      "I895.0" { ExternalVisible := 'False'} : Bool := FALSE;   // I895.0
      "I895.1" { ExternalVisible := 'False'} : Bool := FALSE;   // I895.1
      "I895.2" { ExternalVisible := 'False'} : Bool := FALSE;   // I895.2
      "I895.3" { ExternalVisible := 'False'} : Bool := FALSE;   // I895.3
      "I895.4" { ExternalVisible := 'False'} : Bool := FALSE;   // I895.4
      "I895.5" { ExternalVisible := 'False'} : Bool := FALSE;   // I895.5
      "I895.6" { ExternalVisible := 'False'} : Bool := FALSE;   // I895.6
      "I895.7" { ExternalVisible := 'False'} : Bool := FALSE;   // I895.7
      "I896.0" { ExternalVisible := 'False'} : Bool := FALSE;   // I896.0
      "I896.1" { ExternalVisible := 'False'} : Bool := FALSE;   // I896.1
      "I896.2" { ExternalVisible := 'False'} : Bool := FALSE;   // I896.2
      "I896.3" { ExternalVisible := 'False'} : Bool := FALSE;   // I896.3
      "I896.4" { ExternalVisible := 'False'} : Bool := FALSE;   // I896.4
      "I896.5" { ExternalVisible := 'False'} : Bool := FALSE;   // I896.5
      "I896.6" { ExternalVisible := 'False'} : Bool := FALSE;   // I896.6
      "I896.7" { ExternalVisible := 'False'} : Bool := FALSE;   // I896.7
      "I897.0" { ExternalVisible := 'False'} : Bool := FALSE;   // I897.0
      "I897.1" { ExternalVisible := 'False'} : Bool := FALSE;   // I897.1
      "I897.2" { ExternalVisible := 'False'} : Bool := FALSE;   // I897.2
      "I897.3" { ExternalVisible := 'False'} : Bool := FALSE;   // I897.3
      "I897.4" { ExternalVisible := 'False'} : Bool := FALSE;   // I897.4
      "I897.5" { ExternalVisible := 'False'} : Bool := FALSE;   // I897.5
      "I897.6" { ExternalVisible := 'False'} : Bool := FALSE;   // I897.6
      "I897.7" { ExternalVisible := 'False'} : Bool := FALSE;   // I897.7
      "I898.0" { ExternalVisible := 'False'} : Bool := FALSE;   // I898.0
      "I898.1" { ExternalVisible := 'False'} : Bool := FALSE;   // I898.1
      "I898.2" { ExternalVisible := 'False'} : Bool := FALSE;   // I898.2
      "I898.3" { ExternalVisible := 'False'} : Bool := FALSE;   // I898.3
      "I898.4" { ExternalVisible := 'False'} : Bool := FALSE;   // I898.4
      "I898.5" { ExternalVisible := 'False'} : Bool := FALSE;   // I898.5
      "I898.6" { ExternalVisible := 'False'} : Bool := FALSE;   // I898.6
      "I898.7" { ExternalVisible := 'False'} : Bool := FALSE;   // I898.7
      "I899.0" { ExternalVisible := 'False'} : Bool := FALSE;   // I899.0
      "I899.1" { ExternalVisible := 'False'} : Bool := FALSE;   // I899.1
      "I899.2" { ExternalVisible := 'False'} : Bool := FALSE;   // I899.2
      "I899.3" { ExternalVisible := 'False'} : Bool := FALSE;   // I899.3
      "I899.4" { ExternalVisible := 'False'} : Bool := FALSE;   // I899.4
      "I899.5" { ExternalVisible := 'False'} : Bool := FALSE;   // I899.5
      "I899.6" { ExternalVisible := 'False'} : Bool := FALSE;   // I899.6
      "I899.7" { ExternalVisible := 'False'} : Bool := FALSE;   // I899.7
      "I900.0" { ExternalVisible := 'False'} : Bool := FALSE;   // I900.0
      "I900.1" { ExternalVisible := 'False'} : Bool := FALSE;   // I900.1
      "I900.2" { ExternalVisible := 'False'} : Bool := FALSE;   // I900.2
      "I900.3" { ExternalVisible := 'False'} : Bool := FALSE;   // I900.3
      "I900.4" { ExternalVisible := 'False'} : Bool := FALSE;   // I900.4
      "I900.5" { ExternalVisible := 'False'} : Bool := FALSE;   // I900.5
      "I900.6" { ExternalVisible := 'False'} : Bool := FALSE;   // I900.6
      "I900.7" { ExternalVisible := 'False'} : Bool := FALSE;   // I900.7
   END_VAR
BEGIN
END_DATA_BLOCK

DATA_BLOCK "ST_OUTPUT_Map_DB"   // DB103
{ S7_Optimized_Access := 'FALSE' }
// stored: AutoNumber false
   VAR
      "Q0.0" { ExternalVisible := 'False'} : Bool := FALSE;   // Q0.0
      "Q0.1" { ExternalVisible := 'False'} : Bool := FALSE;   // Q0.1
      "Q0.2" { ExternalVisible := 'False'} : Bool := FALSE;   // Q0.2
      "Q0.3" { ExternalVisible := 'False'} : Bool := FALSE;   // Q0.3
      "Q0.4" { ExternalVisible := 'False'} : Bool := FALSE;   // Q0.4
      "Q0.5" { ExternalVisible := 'False'} : Bool := FALSE;   // Q0.5
      "Q0.6" { ExternalVisible := 'False'} : Bool := FALSE;   // Q0.6
      "Q0.7" { ExternalVisible := 'False'} : Bool := FALSE;   // Q0.7
      "Q1.0" { ExternalVisible := 'False'} : Bool := FALSE;   // Q1.0
      "Q1.1" { ExternalVisible := 'False'} : Bool := FALSE;   // Q1.1
      "Q1.2" { ExternalVisible := 'False'} : Bool := FALSE;   // Q1.2
      "Q1.3" { ExternalVisible := 'False'} : Bool := FALSE;   // Q1.3
      "Q1.4" { ExternalVisible := 'False'} : Bool := FALSE;   // Q1.4
      "Q1.5" { ExternalVisible := 'False'} : Bool := FALSE;   // Q1.5
      "Q1.6" { ExternalVisible := 'False'} : Bool := FALSE;   // Q1.6
      "Q1.7" { ExternalVisible := 'False'} : Bool := FALSE;   // Q1.7
      "Q2.0" { ExternalVisible := 'False'} : Bool := FALSE;   // Q2.0
      "Q2.1" { ExternalVisible := 'False'} : Bool := FALSE;   // Q2.1
      "Q2.2" { ExternalVisible := 'False'} : Bool := FALSE;   // Q2.2
      "Q2.3" { ExternalVisible := 'False'} : Bool := FALSE;   // Q2.3
      "Q2.4" { ExternalVisible := 'False'} : Bool := FALSE;   // Q2.4
      "Q2.5" { ExternalVisible := 'False'} : Bool := FALSE;   // Q2.5
      "Q2.6" { ExternalVisible := 'False'} : Bool := FALSE;   // Q2.6
      "Q2.7" { ExternalVisible := 'False'} : Bool := FALSE;   // Q2.7
      "Q3.0" { ExternalVisible := 'False'} : Bool := FALSE;   // Q3.0
      "Q3.1" { ExternalVisible := 'False'} : Bool := FALSE;   // Q3.1
      "Q3.2" { ExternalVisible := 'False'} : Bool := FALSE;   // Q3.2
      "Q3.3" { ExternalVisible := 'False'} : Bool := FALSE;   // Q3.3
      "Q3.4" { ExternalVisible := 'False'} : Bool := FALSE;   // Q3.4
      "Q3.5" { ExternalVisible := 'False'} : Bool := FALSE;   // Q3.5
      "Q3.6" { ExternalVisible := 'False'} : Bool := FALSE;   // Q3.6
      "Q3.7" { ExternalVisible := 'False'} : Bool := FALSE;   // Q3.7
      "Q4.0" { ExternalVisible := 'False'} : Bool := FALSE;   // Q4.0
      "Q4.1" { ExternalVisible := 'False'} : Bool := FALSE;   // Q4.1
      "Q4.2" { ExternalVisible := 'False'} : Bool := FALSE;   // Q4.2
      "Q4.3" { ExternalVisible := 'False'} : Bool := FALSE;   // Q4.3
      "Q4.4" { ExternalVisible := 'False'} : Bool := FALSE;   // Q4.4
      "Q4.5" { ExternalVisible := 'False'} : Bool := FALSE;   // Q4.5
      "Q4.6" { ExternalVisible := 'False'} : Bool := FALSE;   // Q4.6
      "Q4.7" { ExternalVisible := 'False'} : Bool := FALSE;   // Q4.7
      "Q5.0" { ExternalVisible := 'False'} : Bool := FALSE;   // Q5.0
      "Q5.1" { ExternalVisible := 'False'} : Bool := FALSE;   // Q5.1
      "Q5.2" { ExternalVisible := 'False'} : Bool := FALSE;   // Q5.2
      "Q5.3" { ExternalVisible := 'False'} : Bool := FALSE;   // Q5.3
      "Q5.4" { ExternalVisible := 'False'} : Bool := FALSE;   // Q5.4
      "Q5.5" { ExternalVisible := 'False'} : Bool := FALSE;   // Q5.5
      "Q5.6" { ExternalVisible := 'False'} : Bool := FALSE;   // Q5.6
      "Q5.7" { ExternalVisible := 'False'} : Bool := FALSE;   // Q5.7
      "Q6.0" { ExternalVisible := 'False'} : Bool := FALSE;   // Q6.0
      "Q6.1" { ExternalVisible := 'False'} : Bool := FALSE;   // Q6.1
      "Q6.2" { ExternalVisible := 'False'} : Bool := FALSE;   // Q6.2
      "Q6.3" { ExternalVisible := 'False'} : Bool := FALSE;   // Q6.3
      "Q6.4" { ExternalVisible := 'False'} : Bool := FALSE;   // Q6.4
      "Q6.5" { ExternalVisible := 'False'} : Bool := FALSE;   // Q6.5
      "Q6.6" { ExternalVisible := 'False'} : Bool := FALSE;   // Q6.6
      "Q6.7" { ExternalVisible := 'False'} : Bool := FALSE;   // Q6.7
      "Q7.0" { ExternalVisible := 'False'} : Bool := FALSE;   // Q7.0
      "Q7.1" { ExternalVisible := 'False'} : Bool := FALSE;   // Q7.1
      "Q7.2" { ExternalVisible := 'False'} : Bool := FALSE;   // Q7.2
      "Q7.3" { ExternalVisible := 'False'} : Bool := FALSE;   // Q7.3
      "Q7.4" { ExternalVisible := 'False'} : Bool := FALSE;   // Q7.4
      "Q7.5" { ExternalVisible := 'False'} : Bool := FALSE;   // Q7.5
      "Q7.6" { ExternalVisible := 'False'} : Bool := FALSE;   // Q7.6
      "Q7.7" { ExternalVisible := 'False'} : Bool := FALSE;   // Q7.7
      "Q8.0" { ExternalVisible := 'False'} : Bool := FALSE;   // Q8.0
      "Q8.1" { ExternalVisible := 'False'} : Bool := FALSE;   // Q8.1
      "Q8.2" { ExternalVisible := 'False'} : Bool := FALSE;   // Q8.2
      "Q8.3" { ExternalVisible := 'False'} : Bool := FALSE;   // Q8.3
      "Q8.4" { ExternalVisible := 'False'} : Bool := FALSE;   // Q8.4
      "Q8.5" { ExternalVisible := 'False'} : Bool := FALSE;   // Q8.5
      "Q8.6" { ExternalVisible := 'False'} : Bool := FALSE;   // Q8.6
      "Q8.7" { ExternalVisible := 'False'} : Bool := FALSE;   // Q8.7
      "Q9.0" { ExternalVisible := 'False'} : Bool := FALSE;   // Q9.0
      "Q9.1" { ExternalVisible := 'False'} : Bool := FALSE;   // Q9.1
      "Q9.2" { ExternalVisible := 'False'} : Bool := FALSE;   // Q9.2
      "Q9.3" { ExternalVisible := 'False'} : Bool := FALSE;   // Q9.3
      "Q9.4" { ExternalVisible := 'False'} : Bool := FALSE;   // Q9.4
      "Q9.5" { ExternalVisible := 'False'} : Bool := FALSE;   // Q9.5
      "Q9.6" { ExternalVisible := 'False'} : Bool := FALSE;   // Q9.6
      "Q9.7" { ExternalVisible := 'False'} : Bool := FALSE;   // Q9.7
      PX1 { ExternalVisible := 'False'} : Bool := FALSE;   // 柱灯红色
      PX2 { ExternalVisible := 'False'} : Bool := FALSE;   // 柱灯黄色
      PX3 { ExternalVisible := 'False'} : Bool := FALSE;   // 柱灯蓝色
      PX4 { ExternalVisible := 'False'} : Bool := FALSE;   // 柱灯绿色
      PX5 { ExternalVisible := 'False'} : Bool := FALSE;   // 蜂鸣器
      GBS1_S31 { ExternalVisible := 'False'} : Bool := FALSE;   // 安全门1解锁
      GBS2_S31 { ExternalVisible := 'False'} : Bool := FALSE;   // 安全门2解锁
      "Q10.7" { ExternalVisible := 'False'} : Bool := FALSE;   // Q10.7
      "Q11.0" { ExternalVisible := 'False'} : Bool := FALSE;   // Q11.0
      "Q11.1" { ExternalVisible := 'False'} : Bool := FALSE;   // Q11.1
      "Q11.2" { ExternalVisible := 'False'} : Bool := FALSE;   // Q11.2
      "Q11.3" { ExternalVisible := 'False'} : Bool := FALSE;   // Q11.3
      "Q11.4" { ExternalVisible := 'False'} : Bool := FALSE;   // Q11.4
      "Q11.5" { ExternalVisible := 'False'} : Bool := FALSE;   // Q11.5
      "Q11.6" { ExternalVisible := 'False'} : Bool := FALSE;   // Q11.6
      "Q11.7" { ExternalVisible := 'False'} : Bool := FALSE;   // Q11.7
      "Q12.0" { ExternalVisible := 'False'} : Bool := FALSE;   // Q12.0
      "Q12.1" { ExternalVisible := 'False'} : Bool := FALSE;   // Q12.1
      "Q12.2" { ExternalVisible := 'False'} : Bool := FALSE;   // Q12.2
      "Q12.3" { ExternalVisible := 'False'} : Bool := FALSE;   // Q12.3
      "Q12.4" { ExternalVisible := 'False'} : Bool := FALSE;   // Q12.4
      "Q12.5" { ExternalVisible := 'False'} : Bool := FALSE;   // Q12.5
      "Q12.6" { ExternalVisible := 'False'} : Bool := FALSE;   // Q12.6
      "Q12.7" { ExternalVisible := 'False'} : Bool := FALSE;   // Q12.7
      "Q13.0" { ExternalVisible := 'False'} : Bool := FALSE;   // Q13.0
      "Q13.1" { ExternalVisible := 'False'} : Bool := FALSE;   // Q13.1
      "Q13.2" { ExternalVisible := 'False'} : Bool := FALSE;   // Q13.2
      "Q13.3" { ExternalVisible := 'False'} : Bool := FALSE;   // Q13.3
      "Q13.4" { ExternalVisible := 'False'} : Bool := FALSE;   // Q13.4
      "Q13.5" { ExternalVisible := 'False'} : Bool := FALSE;   // Q13.5
      "Q13.6" { ExternalVisible := 'False'} : Bool := FALSE;   // Q13.6
      "Q13.7" { ExternalVisible := 'False'} : Bool := FALSE;   // Q13.7
      "Q14.0" { ExternalVisible := 'False'} : Bool := FALSE;   // Q14.0
      "Q14.1" { ExternalVisible := 'False'} : Bool := FALSE;   // Q14.1
      "Q14.2" { ExternalVisible := 'False'} : Bool := FALSE;   // Q14.2
      "Q14.3" { ExternalVisible := 'False'} : Bool := FALSE;   // Q14.3
      "Q14.4" { ExternalVisible := 'False'} : Bool := FALSE;   // Q14.4
      "Q14.5" { ExternalVisible := 'False'} : Bool := FALSE;   // Q14.5
      "Q14.6" { ExternalVisible := 'False'} : Bool := FALSE;   // Q14.6
      "Q14.7" { ExternalVisible := 'False'} : Bool := FALSE;   // Q14.7
      "Q15.0" { ExternalVisible := 'False'} : Bool := FALSE;   // Q15.0
      "Q15.1" { ExternalVisible := 'False'} : Bool := FALSE;   // Q15.1
      "Q15.2" { ExternalVisible := 'False'} : Bool := FALSE;   // Q15.2
      "Q15.3" { ExternalVisible := 'False'} : Bool := FALSE;   // Q15.3
      "Q15.4" { ExternalVisible := 'False'} : Bool := FALSE;   // Q15.4
      "Q15.5" { ExternalVisible := 'False'} : Bool := FALSE;   // Q15.5
      "Q15.6" { ExternalVisible := 'False'} : Bool := FALSE;   // Q15.6
      "Q15.7" { ExternalVisible := 'False'} : Bool := FALSE;   // Q15.7
      "Q16.0" { ExternalVisible := 'False'} : Bool := FALSE;   // Q16.0
      "Q16.1" { ExternalVisible := 'False'} : Bool := FALSE;   // Q16.1
      "Q16.2" { ExternalVisible := 'False'} : Bool := FALSE;   // Q16.2
      "Q16.3" { ExternalVisible := 'False'} : Bool := FALSE;   // Q16.3
      "Q16.4" { ExternalVisible := 'False'} : Bool := FALSE;   // Q16.4
      "Q16.5" { ExternalVisible := 'False'} : Bool := FALSE;   // Q16.5
      "Q16.6" { ExternalVisible := 'False'} : Bool := FALSE;   // Q16.6
      "Q16.7" { ExternalVisible := 'False'} : Bool := FALSE;   // Q16.7
      "Q17.0" { ExternalVisible := 'False'} : Bool := FALSE;   // Q17.0
      "Q17.1" { ExternalVisible := 'False'} : Bool := FALSE;   // Q17.1
      "Q17.2" { ExternalVisible := 'False'} : Bool := FALSE;   // Q17.2
      "Q17.3" { ExternalVisible := 'False'} : Bool := FALSE;   // Q17.3
      "Q17.4" { ExternalVisible := 'False'} : Bool := FALSE;   // Q17.4
      "Q17.5" { ExternalVisible := 'False'} : Bool := FALSE;   // Q17.5
      "Q17.6" { ExternalVisible := 'False'} : Bool := FALSE;   // Q17.6
      "Q17.7" { ExternalVisible := 'False'} : Bool := FALSE;   // Q17.7
      "Q18.0" { ExternalVisible := 'False'} : Bool := FALSE;   // Q18.0
      "Q18.1" { ExternalVisible := 'False'} : Bool := FALSE;   // Q18.1
      "Q18.2" { ExternalVisible := 'False'} : Bool := FALSE;   // Q18.2
      "Q18.3" { ExternalVisible := 'False'} : Bool := FALSE;   // Q18.3
      "Q18.4" { ExternalVisible := 'False'} : Bool := FALSE;   // Q18.4
      "Q18.5" { ExternalVisible := 'False'} : Bool := FALSE;   // Q18.5
      "Q18.6" { ExternalVisible := 'False'} : Bool := FALSE;   // Q18.6
      "Q18.7" { ExternalVisible := 'False'} : Bool := FALSE;   // Q18.7
      "Q19.0" { ExternalVisible := 'False'} : Bool := FALSE;   // Q19.0
      "Q19.1" { ExternalVisible := 'False'} : Bool := FALSE;   // Q19.1
      "Q19.2" { ExternalVisible := 'False'} : Bool := FALSE;   // Q19.2
      "Q19.3" { ExternalVisible := 'False'} : Bool := FALSE;   // Q19.3
      "Q19.4" { ExternalVisible := 'False'} : Bool := FALSE;   // Q19.4
      "Q19.5" { ExternalVisible := 'False'} : Bool := FALSE;   // Q19.5
      "Q19.6" { ExternalVisible := 'False'} : Bool := FALSE;   // Q19.6
      "Q19.7" { ExternalVisible := 'False'} : Bool := FALSE;   // Q19.7
      "Q20.0" { ExternalVisible := 'False'} : Bool := FALSE;   // Q20.0
      "Q20.1" { ExternalVisible := 'False'} : Bool := FALSE;   // Q20.1
      "Q20.2" { ExternalVisible := 'False'} : Bool := FALSE;   // Q20.2
      "Q20.3" { ExternalVisible := 'False'} : Bool := FALSE;   // Q20.3
      "Q20.4" { ExternalVisible := 'False'} : Bool := FALSE;   // Q20.4
      "Q20.5" { ExternalVisible := 'False'} : Bool := FALSE;   // Q20.5
      "Q20.6" { ExternalVisible := 'False'} : Bool := FALSE;   // Q20.6
      "Q20.7" { ExternalVisible := 'False'} : Bool := FALSE;   // Q20.7
      "Q21.0" { ExternalVisible := 'False'} : Bool := FALSE;   // Q21.0
      "Q21.1" { ExternalVisible := 'False'} : Bool := FALSE;   // Q21.1
      "Q21.2" { ExternalVisible := 'False'} : Bool := FALSE;   // Q21.2
      "Q21.3" { ExternalVisible := 'False'} : Bool := FALSE;   // Q21.3
      "Q21.4" { ExternalVisible := 'False'} : Bool := FALSE;   // Q21.4
      "Q21.5" { ExternalVisible := 'False'} : Bool := FALSE;   // Q21.5
      "Q21.6" { ExternalVisible := 'False'} : Bool := FALSE;   // Q21.6
      "Q21.7" { ExternalVisible := 'False'} : Bool := FALSE;   // Q21.7
      "Q22.0" { ExternalVisible := 'False'} : Bool := FALSE;   // Q22.0
      "Q22.1" { ExternalVisible := 'False'} : Bool := FALSE;   // Q22.1
      "Q22.2" { ExternalVisible := 'False'} : Bool := FALSE;   // Q22.2
      "Q22.3" { ExternalVisible := 'False'} : Bool := FALSE;   // Q22.3
      "Q22.4" { ExternalVisible := 'False'} : Bool := FALSE;   // Q22.4
      "Q22.5" { ExternalVisible := 'False'} : Bool := FALSE;   // Q22.5
      "Q22.6" { ExternalVisible := 'False'} : Bool := FALSE;   // Q22.6
      "Q22.7" { ExternalVisible := 'False'} : Bool := FALSE;   // Q22.7
      "Q23.0" { ExternalVisible := 'False'} : Bool := FALSE;   // Q23.0
      "Q23.1" { ExternalVisible := 'False'} : Bool := FALSE;   // Q23.1
      "Q23.2" { ExternalVisible := 'False'} : Bool := FALSE;   // Q23.2
      "Q23.3" { ExternalVisible := 'False'} : Bool := FALSE;   // Q23.3
      "Q23.4" { ExternalVisible := 'False'} : Bool := FALSE;   // Q23.4
      "Q23.5" { ExternalVisible := 'False'} : Bool := FALSE;   // Q23.5
      "Q23.6" { ExternalVisible := 'False'} : Bool := FALSE;   // Q23.6
      "Q23.7" { ExternalVisible := 'False'} : Bool := FALSE;   // Q23.7
      "Q24.0" { ExternalVisible := 'False'} : Bool := FALSE;   // Q24.0
      "Q24.1" { ExternalVisible := 'False'} : Bool := FALSE;   // Q24.1
      "Q24.2" { ExternalVisible := 'False'} : Bool := FALSE;   // Q24.2
      "Q24.3" { ExternalVisible := 'False'} : Bool := FALSE;   // Q24.3
      "Q24.4" { ExternalVisible := 'False'} : Bool := FALSE;   // Q24.4
      "Q24.5" { ExternalVisible := 'False'} : Bool := FALSE;   // Q24.5
      "Q24.6" { ExternalVisible := 'False'} : Bool := FALSE;   // Q24.6
      "Q24.7" { ExternalVisible := 'False'} : Bool := FALSE;   // Q24.7
      "Q25.0" { ExternalVisible := 'False'} : Bool := FALSE;   // Q25.0
      "Q25.1" { ExternalVisible := 'False'} : Bool := FALSE;   // Q25.1
      "Q25.2" { ExternalVisible := 'False'} : Bool := FALSE;   // Q25.2
      "Q25.3" { ExternalVisible := 'False'} : Bool := FALSE;   // Q25.3
      "Q25.4" { ExternalVisible := 'False'} : Bool := FALSE;   // Q25.4
      "Q25.5" { ExternalVisible := 'False'} : Bool := FALSE;   // Q25.5
      "Q25.6" { ExternalVisible := 'False'} : Bool := FALSE;   // Q25.6
      "Q25.7" { ExternalVisible := 'False'} : Bool := FALSE;   // Q25.7
      "Q26.0" { ExternalVisible := 'False'} : Bool := FALSE;   // Q26.0
      "Q26.1" { ExternalVisible := 'False'} : Bool := FALSE;   // Q26.1
      "Q26.2" { ExternalVisible := 'False'} : Bool := FALSE;   // Q26.2
      "Q26.3" { ExternalVisible := 'False'} : Bool := FALSE;   // Q26.3
      "Q26.4" { ExternalVisible := 'False'} : Bool := FALSE;   // Q26.4
      "Q26.5" { ExternalVisible := 'False'} : Bool := FALSE;   // Q26.5
      "Q26.6" { ExternalVisible := 'False'} : Bool := FALSE;   // Q26.6
      "Q26.7" { ExternalVisible := 'False'} : Bool := FALSE;   // Q26.7
      "Q27.0" { ExternalVisible := 'False'} : Bool := FALSE;   // Q27.0
      "Q27.1" { ExternalVisible := 'False'} : Bool := FALSE;   // Q27.1
      "Q27.2" { ExternalVisible := 'False'} : Bool := FALSE;   // Q27.2
      "Q27.3" { ExternalVisible := 'False'} : Bool := FALSE;   // Q27.3
      "Q27.4" { ExternalVisible := 'False'} : Bool := FALSE;   // Q27.4
      "Q27.5" { ExternalVisible := 'False'} : Bool := FALSE;   // Q27.5
      "Q27.6" { ExternalVisible := 'False'} : Bool := FALSE;   // Q27.6
      "Q27.7" { ExternalVisible := 'False'} : Bool := FALSE;   // Q27.7
      "Q28.0" { ExternalVisible := 'False'} : Bool := FALSE;   // Q28.0
      "Q28.1" { ExternalVisible := 'False'} : Bool := FALSE;   // Q28.1
      "Q28.2" { ExternalVisible := 'False'} : Bool := FALSE;   // Q28.2
      "Q28.3" { ExternalVisible := 'False'} : Bool := FALSE;   // Q28.3
      "Q28.4" { ExternalVisible := 'False'} : Bool := FALSE;   // Q28.4
      "Q28.5" { ExternalVisible := 'False'} : Bool := FALSE;   // Q28.5
      "Q28.6" { ExternalVisible := 'False'} : Bool := FALSE;   // Q28.6
      "Q28.7" { ExternalVisible := 'False'} : Bool := FALSE;   // Q28.7
      "Q29.0" { ExternalVisible := 'False'} : Bool := FALSE;   // Q29.0
      "Q29.1" { ExternalVisible := 'False'} : Bool := FALSE;   // Q29.1
      "Q29.2" { ExternalVisible := 'False'} : Bool := FALSE;   // Q29.2
      "Q29.3" { ExternalVisible := 'False'} : Bool := FALSE;   // Q29.3
      "Q29.4" { ExternalVisible := 'False'} : Bool := FALSE;   // Q29.4
      "Q29.5" { ExternalVisible := 'False'} : Bool := FALSE;   // Q29.5
      "Q29.6" { ExternalVisible := 'False'} : Bool := FALSE;   // Q29.6
      "Q29.7" { ExternalVisible := 'False'} : Bool := FALSE;   // Q29.7
      "Q30.0" { ExternalVisible := 'False'} : Bool := FALSE;   // Q30.0
      "Q30.1" { ExternalVisible := 'False'} : Bool := FALSE;   // Q30.1
      "Q30.2" { ExternalVisible := 'False'} : Bool := FALSE;   // Q30.2
      "Q30.3" { ExternalVisible := 'False'} : Bool := FALSE;   // Q30.3
      "Q30.4" { ExternalVisible := 'False'} : Bool := FALSE;   // Q30.4
      "Q30.5" { ExternalVisible := 'False'} : Bool := FALSE;   // Q30.5
      "Q30.6" { ExternalVisible := 'False'} : Bool := FALSE;   // Q30.6
      "Q30.7" { ExternalVisible := 'False'} : Bool := FALSE;   // Q30.7
      "Q31.0" { ExternalVisible := 'False'} : Bool := FALSE;   // Q31.0
      "Q31.1" { ExternalVisible := 'False'} : Bool := FALSE;   // Q31.1
      "Q31.2" { ExternalVisible := 'False'} : Bool := FALSE;   // Q31.2
      "Q31.3" { ExternalVisible := 'False'} : Bool := FALSE;   // Q31.3
      "Q31.4" { ExternalVisible := 'False'} : Bool := FALSE;   // Q31.4
      "Q31.5" { ExternalVisible := 'False'} : Bool := FALSE;   // Q31.5
      "Q31.6" { ExternalVisible := 'False'} : Bool := FALSE;   // Q31.6
      "Q31.7" { ExternalVisible := 'False'} : Bool := FALSE;   // Q31.7
      "Q32.0" { ExternalVisible := 'False'} : Bool := FALSE;   // Q32.0
      "Q32.1" { ExternalVisible := 'False'} : Bool := FALSE;   // Q32.1
      "Q32.2" { ExternalVisible := 'False'} : Bool := FALSE;   // Q32.2
      "Q32.3" { ExternalVisible := 'False'} : Bool := FALSE;   // Q32.3
      "Q32.4" { ExternalVisible := 'False'} : Bool := FALSE;   // Q32.4
      "Q32.5" { ExternalVisible := 'False'} : Bool := FALSE;   // Q32.5
      "Q32.6" { ExternalVisible := 'False'} : Bool := FALSE;   // Q32.6
      "Q32.7" { ExternalVisible := 'False'} : Bool := FALSE;   // Q32.7
      "Q33.0" { ExternalVisible := 'False'} : Bool := FALSE;   // Q33.0
      "Q33.1" { ExternalVisible := 'False'} : Bool := FALSE;   // Q33.1
      "Q33.2" { ExternalVisible := 'False'} : Bool := FALSE;   // Q33.2
      "Q33.3" { ExternalVisible := 'False'} : Bool := FALSE;   // Q33.3
      "Q33.4" { ExternalVisible := 'False'} : Bool := FALSE;   // Q33.4
      "Q33.5" { ExternalVisible := 'False'} : Bool := FALSE;   // Q33.5
      "Q33.6" { ExternalVisible := 'False'} : Bool := FALSE;   // Q33.6
      "Q33.7" { ExternalVisible := 'False'} : Bool := FALSE;   // Q33.7
      "Q34.0" { ExternalVisible := 'False'} : Bool := FALSE;   // Q34.0
      "Q34.1" { ExternalVisible := 'False'} : Bool := FALSE;   // Q34.1
      "Q34.2" { ExternalVisible := 'False'} : Bool := FALSE;   // Q34.2
      "Q34.3" { ExternalVisible := 'False'} : Bool := FALSE;   // Q34.3
      "Q34.4" { ExternalVisible := 'False'} : Bool := FALSE;   // Q34.4
      "Q34.5" { ExternalVisible := 'False'} : Bool := FALSE;   // Q34.5
      "Q34.6" { ExternalVisible := 'False'} : Bool := FALSE;   // Q34.6
      "Q34.7" { ExternalVisible := 'False'} : Bool := FALSE;   // Q34.7
      "Q35.0" { ExternalVisible := 'False'} : Bool := FALSE;   // Q35.0
      "Q35.1" { ExternalVisible := 'False'} : Bool := FALSE;   // Q35.1
      "Q35.2" { ExternalVisible := 'False'} : Bool := FALSE;   // Q35.2
      "Q35.3" { ExternalVisible := 'False'} : Bool := FALSE;   // Q35.3
      "Q35.4" { ExternalVisible := 'False'} : Bool := FALSE;   // Q35.4
      "Q35.5" { ExternalVisible := 'False'} : Bool := FALSE;   // Q35.5
      "Q35.6" { ExternalVisible := 'False'} : Bool := FALSE;   // Q35.6
      "Q35.7" { ExternalVisible := 'False'} : Bool := FALSE;   // Q35.7
      "Q36.0" { ExternalVisible := 'False'} : Bool := FALSE;   // Q36.0
      "Q36.1" { ExternalVisible := 'False'} : Bool := FALSE;   // Q36.1
      "Q36.2" { ExternalVisible := 'False'} : Bool := FALSE;   // Q36.2
      "Q36.3" { ExternalVisible := 'False'} : Bool := FALSE;   // Q36.3
      "Q36.4" { ExternalVisible := 'False'} : Bool := FALSE;   // Q36.4
      "Q36.5" { ExternalVisible := 'False'} : Bool := FALSE;   // Q36.5
      "Q36.6" { ExternalVisible := 'False'} : Bool := FALSE;   // Q36.6
      "Q36.7" { ExternalVisible := 'False'} : Bool := FALSE;   // Q36.7
      "Q37.0" { ExternalVisible := 'False'} : Bool := FALSE;   // Q37.0
      "Q37.1" { ExternalVisible := 'False'} : Bool := FALSE;   // Q37.1
      "Q37.2" { ExternalVisible := 'False'} : Bool := FALSE;   // Q37.2
      "Q37.3" { ExternalVisible := 'False'} : Bool := FALSE;   // Q37.3
      "Q37.4" { ExternalVisible := 'False'} : Bool := FALSE;   // Q37.4
      "Q37.5" { ExternalVisible := 'False'} : Bool := FALSE;   // Q37.5
      "Q37.6" { ExternalVisible := 'False'} : Bool := FALSE;   // Q37.6
      "Q37.7" { ExternalVisible := 'False'} : Bool := FALSE;   // Q37.7
      "Q38.0" { ExternalVisible := 'False'} : Bool := FALSE;   // Q38.0
      "Q38.1" { ExternalVisible := 'False'} : Bool := FALSE;   // Q38.1
      "Q38.2" { ExternalVisible := 'False'} : Bool := FALSE;   // Q38.2
      "Q38.3" { ExternalVisible := 'False'} : Bool := FALSE;   // Q38.3
      "Q38.4" { ExternalVisible := 'False'} : Bool := FALSE;   // Q38.4
      "Q38.5" { ExternalVisible := 'False'} : Bool := FALSE;   // Q38.5
      "Q38.6" { ExternalVisible := 'False'} : Bool := FALSE;   // Q38.6
      "Q38.7" { ExternalVisible := 'False'} : Bool := FALSE;   // Q38.7
      "Q39.0" { ExternalVisible := 'False'} : Bool := FALSE;   // Q39.0
      "Q39.1" { ExternalVisible := 'False'} : Bool := FALSE;   // Q39.1
      "Q39.2" { ExternalVisible := 'False'} : Bool := FALSE;   // Q39.2
      "Q39.3" { ExternalVisible := 'False'} : Bool := FALSE;   // Q39.3
      "Q39.4" { ExternalVisible := 'False'} : Bool := FALSE;   // Q39.4
      "Q39.5" { ExternalVisible := 'False'} : Bool := FALSE;   // Q39.5
      "Q39.6" { ExternalVisible := 'False'} : Bool := FALSE;   // Q39.6
      "Q39.7" { ExternalVisible := 'False'} : Bool := FALSE;   // Q39.7
      "Q40.0" { ExternalVisible := 'False'} : Bool := FALSE;   // Q40.0
      "Q40.1" { ExternalVisible := 'False'} : Bool := FALSE;   // Q40.1
      "Q40.2" { ExternalVisible := 'False'} : Bool := FALSE;   // Q40.2
      "Q40.3" { ExternalVisible := 'False'} : Bool := FALSE;   // Q40.3
      "Q40.4" { ExternalVisible := 'False'} : Bool := FALSE;   // Q40.4
      "Q40.5" { ExternalVisible := 'False'} : Bool := FALSE;   // Q40.5
      "Q40.6" { ExternalVisible := 'False'} : Bool := FALSE;   // Q40.6
      "Q40.7" { ExternalVisible := 'False'} : Bool := FALSE;   // Q40.7
      "Q41.0" { ExternalVisible := 'False'} : Bool := FALSE;   // Q41.0
      "Q41.1" { ExternalVisible := 'False'} : Bool := FALSE;   // Q41.1
      "Q41.2" { ExternalVisible := 'False'} : Bool := FALSE;   // Q41.2
      "Q41.3" { ExternalVisible := 'False'} : Bool := FALSE;   // Q41.3
      "Q41.4" { ExternalVisible := 'False'} : Bool := FALSE;   // Q41.4
      "Q41.5" { ExternalVisible := 'False'} : Bool := FALSE;   // Q41.5
      "Q41.6" { ExternalVisible := 'False'} : Bool := FALSE;   // Q41.6
      "Q41.7" { ExternalVisible := 'False'} : Bool := FALSE;   // Q41.7
      "Q42.0" { ExternalVisible := 'False'} : Bool := FALSE;   // Q42.0
      "Q42.1" { ExternalVisible := 'False'} : Bool := FALSE;   // Q42.1
      "Q42.2" { ExternalVisible := 'False'} : Bool := FALSE;   // Q42.2
      "Q42.3" { ExternalVisible := 'False'} : Bool := FALSE;   // Q42.3
      "Q42.4" { ExternalVisible := 'False'} : Bool := FALSE;   // Q42.4
      "Q42.5" { ExternalVisible := 'False'} : Bool := FALSE;   // Q42.5
      "Q42.6" { ExternalVisible := 'False'} : Bool := FALSE;   // Q42.6
      "Q42.7" { ExternalVisible := 'False'} : Bool := FALSE;   // Q42.7
      "Q43.0" { ExternalVisible := 'False'} : Bool := FALSE;   // Q43.0
      "Q43.1" { ExternalVisible := 'False'} : Bool := FALSE;   // Q43.1
      "Q43.2" { ExternalVisible := 'False'} : Bool := FALSE;   // Q43.2
      "Q43.3" { ExternalVisible := 'False'} : Bool := FALSE;   // Q43.3
      "Q43.4" { ExternalVisible := 'False'} : Bool := FALSE;   // Q43.4
      "Q43.5" { ExternalVisible := 'False'} : Bool := FALSE;   // Q43.5
      "Q43.6" { ExternalVisible := 'False'} : Bool := FALSE;   // Q43.6
      "Q43.7" { ExternalVisible := 'False'} : Bool := FALSE;   // Q43.7
      "Q44.0" { ExternalVisible := 'False'} : Bool := FALSE;   // Q44.0
      "Q44.1" { ExternalVisible := 'False'} : Bool := FALSE;   // Q44.1
      "Q44.2" { ExternalVisible := 'False'} : Bool := FALSE;   // Q44.2
      "Q44.3" { ExternalVisible := 'False'} : Bool := FALSE;   // Q44.3
      "Q44.4" { ExternalVisible := 'False'} : Bool := FALSE;   // Q44.4
      "Q44.5" { ExternalVisible := 'False'} : Bool := FALSE;   // Q44.5
      "Q44.6" { ExternalVisible := 'False'} : Bool := FALSE;   // Q44.6
      "Q44.7" { ExternalVisible := 'False'} : Bool := FALSE;   // Q44.7
      "Q45.0" { ExternalVisible := 'False'} : Bool := FALSE;   // Q45.0
      "Q45.1" { ExternalVisible := 'False'} : Bool := FALSE;   // Q45.1
      "Q45.2" { ExternalVisible := 'False'} : Bool := FALSE;   // Q45.2
      "Q45.3" { ExternalVisible := 'False'} : Bool := FALSE;   // Q45.3
      "Q45.4" { ExternalVisible := 'False'} : Bool := FALSE;   // Q45.4
      "Q45.5" { ExternalVisible := 'False'} : Bool := FALSE;   // Q45.5
      "Q45.6" { ExternalVisible := 'False'} : Bool := FALSE;   // Q45.6
      "Q45.7" { ExternalVisible := 'False'} : Bool := FALSE;   // Q45.7
      "Q46.0" { ExternalVisible := 'False'} : Bool := FALSE;   // Q46.0
      "Q46.1" { ExternalVisible := 'False'} : Bool := FALSE;   // Q46.1
      "Q46.2" { ExternalVisible := 'False'} : Bool := FALSE;   // Q46.2
      "Q46.3" { ExternalVisible := 'False'} : Bool := FALSE;   // Q46.3
      "Q46.4" { ExternalVisible := 'False'} : Bool := FALSE;   // Q46.4
      "Q46.5" { ExternalVisible := 'False'} : Bool := FALSE;   // Q46.5
      "Q46.6" { ExternalVisible := 'False'} : Bool := FALSE;   // Q46.6
      "Q46.7" { ExternalVisible := 'False'} : Bool := FALSE;   // Q46.7
      "Q47.0" { ExternalVisible := 'False'} : Bool := FALSE;   // Q47.0
      "Q47.1" { ExternalVisible := 'False'} : Bool := FALSE;   // Q47.1
      "Q47.2" { ExternalVisible := 'False'} : Bool := FALSE;   // Q47.2
      "Q47.3" { ExternalVisible := 'False'} : Bool := FALSE;   // Q47.3
      "Q47.4" { ExternalVisible := 'False'} : Bool := FALSE;   // Q47.4
      "Q47.5" { ExternalVisible := 'False'} : Bool := FALSE;   // Q47.5
      "Q47.6" { ExternalVisible := 'False'} : Bool := FALSE;   // Q47.6
      "Q47.7" { ExternalVisible := 'False'} : Bool := FALSE;   // Q47.7
      "Q48.0" { ExternalVisible := 'False'} : Bool := FALSE;   // Q48.0
      "Q48.1" { ExternalVisible := 'False'} : Bool := FALSE;   // Q48.1
      "Q48.2" { ExternalVisible := 'False'} : Bool := FALSE;   // Q48.2
      "Q48.3" { ExternalVisible := 'False'} : Bool := FALSE;   // Q48.3
      "Q48.4" { ExternalVisible := 'False'} : Bool := FALSE;   // Q48.4
      "Q48.5" { ExternalVisible := 'False'} : Bool := FALSE;   // Q48.5
      "Q48.6" { ExternalVisible := 'False'} : Bool := FALSE;   // Q48.6
      "Q48.7" { ExternalVisible := 'False'} : Bool := FALSE;   // Q48.7
      "Q49.0" { ExternalVisible := 'False'} : Bool := FALSE;   // Q49.0
      "Q49.1" { ExternalVisible := 'False'} : Bool := FALSE;   // Q49.1
      "Q49.2" { ExternalVisible := 'False'} : Bool := FALSE;   // Q49.2
      "Q49.3" { ExternalVisible := 'False'} : Bool := FALSE;   // Q49.3
      "Q49.4" { ExternalVisible := 'False'} : Bool := FALSE;   // Q49.4
      "Q49.5" { ExternalVisible := 'False'} : Bool := FALSE;   // Q49.5
      "Q49.6" { ExternalVisible := 'False'} : Bool := FALSE;   // Q49.6
      "Q49.7" { ExternalVisible := 'False'} : Bool := FALSE;   // Q49.7
      "Q50.0" { ExternalVisible := 'False'} : Bool := FALSE;   // Q50.0
      "Q50.1" { ExternalVisible := 'False'} : Bool := FALSE;   // Q50.1
      "Q50.2" { ExternalVisible := 'False'} : Bool := FALSE;   // Q50.2
      "Q50.3" { ExternalVisible := 'False'} : Bool := FALSE;   // Q50.3
      "Q50.4" { ExternalVisible := 'False'} : Bool := FALSE;   // Q50.4
      "Q50.5" { ExternalVisible := 'False'} : Bool := FALSE;   // Q50.5
      "Q50.6" { ExternalVisible := 'False'} : Bool := FALSE;   // Q50.6
      "Q50.7" { ExternalVisible := 'False'} : Bool := FALSE;   // Q50.7
      "Q51.0" { ExternalVisible := 'False'} : Bool := FALSE;   // Q51.0
      "Q51.1" { ExternalVisible := 'False'} : Bool := FALSE;   // Q51.1
      "Q51.2" { ExternalVisible := 'False'} : Bool := FALSE;   // Q51.2
      "Q51.3" { ExternalVisible := 'False'} : Bool := FALSE;   // Q51.3
      "Q51.4" { ExternalVisible := 'False'} : Bool := FALSE;   // Q51.4
      "Q51.5" { ExternalVisible := 'False'} : Bool := FALSE;   // Q51.5
      "Q51.6" { ExternalVisible := 'False'} : Bool := FALSE;   // Q51.6
      "Q51.7" { ExternalVisible := 'False'} : Bool := FALSE;   // Q51.7
      "Q52.0" { ExternalVisible := 'False'} : Bool := FALSE;   // Q52.0
      "Q52.1" { ExternalVisible := 'False'} : Bool := FALSE;   // Q52.1
      "Q52.2" { ExternalVisible := 'False'} : Bool := FALSE;   // Q52.2
      "Q52.3" { ExternalVisible := 'False'} : Bool := FALSE;   // Q52.3
      "Q52.4" { ExternalVisible := 'False'} : Bool := FALSE;   // Q52.4
      "Q52.5" { ExternalVisible := 'False'} : Bool := FALSE;   // Q52.5
      "Q52.6" { ExternalVisible := 'False'} : Bool := FALSE;   // Q52.6
      "Q52.7" { ExternalVisible := 'False'} : Bool := FALSE;   // Q52.7
      "Q53.0" { ExternalVisible := 'False'} : Bool := FALSE;   // Q53.0
      "Q53.1" { ExternalVisible := 'False'} : Bool := FALSE;   // Q53.1
      "Q53.2" { ExternalVisible := 'False'} : Bool := FALSE;   // Q53.2
      "Q53.3" { ExternalVisible := 'False'} : Bool := FALSE;   // Q53.3
      "Q53.4" { ExternalVisible := 'False'} : Bool := FALSE;   // Q53.4
      "Q53.5" { ExternalVisible := 'False'} : Bool := FALSE;   // Q53.5
      "Q53.6" { ExternalVisible := 'False'} : Bool := FALSE;   // Q53.6
      "Q53.7" { ExternalVisible := 'False'} : Bool := FALSE;   // Q53.7
      "Q54.0" { ExternalVisible := 'False'} : Bool := FALSE;   // Q54.0
      "Q54.1" { ExternalVisible := 'False'} : Bool := FALSE;   // Q54.1
      "Q54.2" { ExternalVisible := 'False'} : Bool := FALSE;   // Q54.2
      "Q54.3" { ExternalVisible := 'False'} : Bool := FALSE;   // Q54.3
      "Q54.4" { ExternalVisible := 'False'} : Bool := FALSE;   // Q54.4
      "Q54.5" { ExternalVisible := 'False'} : Bool := FALSE;   // Q54.5
      "Q54.6" { ExternalVisible := 'False'} : Bool := FALSE;   // Q54.6
      "Q54.7" { ExternalVisible := 'False'} : Bool := FALSE;   // Q54.7
      "Q55.0" { ExternalVisible := 'False'} : Bool := FALSE;   // Q55.0
      "Q55.1" { ExternalVisible := 'False'} : Bool := FALSE;   // Q55.1
      "Q55.2" { ExternalVisible := 'False'} : Bool := FALSE;   // Q55.2
      "Q55.3" { ExternalVisible := 'False'} : Bool := FALSE;   // Q55.3
      "Q55.4" { ExternalVisible := 'False'} : Bool := FALSE;   // Q55.4
      "Q55.5" { ExternalVisible := 'False'} : Bool := FALSE;   // Q55.5
      "Q55.6" { ExternalVisible := 'False'} : Bool := FALSE;   // Q55.6
      "Q55.7" { ExternalVisible := 'False'} : Bool := FALSE;   // Q55.7
      "Q56.0" { ExternalVisible := 'False'} : Bool := FALSE;   // Q56.0
      "Q56.1" { ExternalVisible := 'False'} : Bool := FALSE;   // Q56.1
      "Q56.2" { ExternalVisible := 'False'} : Bool := FALSE;   // Q56.2
      "Q56.3" { ExternalVisible := 'False'} : Bool := FALSE;   // Q56.3
      "Q56.4" { ExternalVisible := 'False'} : Bool := FALSE;   // Q56.4
      "Q56.5" { ExternalVisible := 'False'} : Bool := FALSE;   // Q56.5
      "Q56.6" { ExternalVisible := 'False'} : Bool := FALSE;   // Q56.6
      "Q56.7" { ExternalVisible := 'False'} : Bool := FALSE;   // Q56.7
      "Q57.0" { ExternalVisible := 'False'} : Bool := FALSE;   // Q57.0
      "Q57.1" { ExternalVisible := 'False'} : Bool := FALSE;   // Q57.1
      "Q57.2" { ExternalVisible := 'False'} : Bool := FALSE;   // Q57.2
      "Q57.3" { ExternalVisible := 'False'} : Bool := FALSE;   // Q57.3
      "Q57.4" { ExternalVisible := 'False'} : Bool := FALSE;   // Q57.4
      "Q57.5" { ExternalVisible := 'False'} : Bool := FALSE;   // Q57.5
      "Q57.6" { ExternalVisible := 'False'} : Bool := FALSE;   // Q57.6
      "Q57.7" { ExternalVisible := 'False'} : Bool := FALSE;   // Q57.7
      "Q58.0" { ExternalVisible := 'False'} : Bool := FALSE;   // Q58.0
      "Q58.1" { ExternalVisible := 'False'} : Bool := FALSE;   // Q58.1
      "Q58.2" { ExternalVisible := 'False'} : Bool := FALSE;   // Q58.2
      "Q58.3" { ExternalVisible := 'False'} : Bool := FALSE;   // Q58.3
      "Q58.4" { ExternalVisible := 'False'} : Bool := FALSE;   // Q58.4
      "Q58.5" { ExternalVisible := 'False'} : Bool := FALSE;   // Q58.5
      "Q58.6" { ExternalVisible := 'False'} : Bool := FALSE;   // Q58.6
      "Q58.7" { ExternalVisible := 'False'} : Bool := FALSE;   // Q58.7
      "Q59.0" { ExternalVisible := 'False'} : Bool := FALSE;   // Q59.0
      "Q59.1" { ExternalVisible := 'False'} : Bool := FALSE;   // Q59.1
      "Q59.2" { ExternalVisible := 'False'} : Bool := FALSE;   // Q59.2
      "Q59.3" { ExternalVisible := 'False'} : Bool := FALSE;   // Q59.3
      "Q59.4" { ExternalVisible := 'False'} : Bool := FALSE;   // Q59.4
      "Q59.5" { ExternalVisible := 'False'} : Bool := FALSE;   // Q59.5
      "Q59.6" { ExternalVisible := 'False'} : Bool := FALSE;   // Q59.6
      "Q59.7" { ExternalVisible := 'False'} : Bool := FALSE;   // Q59.7
      "Q60.0" { ExternalVisible := 'False'} : Bool := FALSE;   // Q60.0
      "Q60.1" { ExternalVisible := 'False'} : Bool := FALSE;   // Q60.1
      "Q60.2" { ExternalVisible := 'False'} : Bool := FALSE;   // Q60.2
      "Q60.3" { ExternalVisible := 'False'} : Bool := FALSE;   // Q60.3
      "Q60.4" { ExternalVisible := 'False'} : Bool := FALSE;   // Q60.4
      "Q60.5" { ExternalVisible := 'False'} : Bool := FALSE;   // Q60.5
      "Q60.6" { ExternalVisible := 'False'} : Bool := FALSE;   // Q60.6
      "Q60.7" { ExternalVisible := 'False'} : Bool := FALSE;   // Q60.7
      "Q61.0" { ExternalVisible := 'False'} : Bool := FALSE;   // Q61.0
      "Q61.1" { ExternalVisible := 'False'} : Bool := FALSE;   // Q61.1
      "Q61.2" { ExternalVisible := 'False'} : Bool := FALSE;   // Q61.2
      "Q61.3" { ExternalVisible := 'False'} : Bool := FALSE;   // Q61.3
      "Q61.4" { ExternalVisible := 'False'} : Bool := FALSE;   // Q61.4
      "Q61.5" { ExternalVisible := 'False'} : Bool := FALSE;   // Q61.5
      "Q61.6" { ExternalVisible := 'False'} : Bool := FALSE;   // Q61.6
      "Q61.7" { ExternalVisible := 'False'} : Bool := FALSE;   // Q61.7
      "Q62.0" { ExternalVisible := 'False'} : Bool := FALSE;   // Q62.0
      "Q62.1" { ExternalVisible := 'False'} : Bool := FALSE;   // Q62.1
      "Q62.2" { ExternalVisible := 'False'} : Bool := FALSE;   // Q62.2
      "Q62.3" { ExternalVisible := 'False'} : Bool := FALSE;   // Q62.3
      "Q62.4" { ExternalVisible := 'False'} : Bool := FALSE;   // Q62.4
      "Q62.5" { ExternalVisible := 'False'} : Bool := FALSE;   // Q62.5
      "Q62.6" { ExternalVisible := 'False'} : Bool := FALSE;   // Q62.6
      "Q62.7" { ExternalVisible := 'False'} : Bool := FALSE;   // Q62.7
      "Q63.0" { ExternalVisible := 'False'} : Bool := FALSE;   // Q63.0
      "Q63.1" { ExternalVisible := 'False'} : Bool := FALSE;   // Q63.1
      "Q63.2" { ExternalVisible := 'False'} : Bool := FALSE;   // Q63.2
      "Q63.3" { ExternalVisible := 'False'} : Bool := FALSE;   // Q63.3
      "Q63.4" { ExternalVisible := 'False'} : Bool := FALSE;   // Q63.4
      "Q63.5" { ExternalVisible := 'False'} : Bool := FALSE;   // Q63.5
      "Q63.6" { ExternalVisible := 'False'} : Bool := FALSE;   // Q63.6
      "Q63.7" { ExternalVisible := 'False'} : Bool := FALSE;   // Q63.7
      "Q64.0" { ExternalVisible := 'False'} : Bool := FALSE;   // Q64.0
      "Q64.1" { ExternalVisible := 'False'} : Bool := FALSE;   // Q64.1
      "Q64.2" { ExternalVisible := 'False'} : Bool := FALSE;   // Q64.2
      "Q64.3" { ExternalVisible := 'False'} : Bool := FALSE;   // Q64.3
      "Q64.4" { ExternalVisible := 'False'} : Bool := FALSE;   // Q64.4
      "Q64.5" { ExternalVisible := 'False'} : Bool := FALSE;   // Q64.5
      "Q64.6" { ExternalVisible := 'False'} : Bool := FALSE;   // Q64.6
      "Q64.7" { ExternalVisible := 'False'} : Bool := FALSE;   // Q64.7
      "Q65.0" { ExternalVisible := 'False'} : Bool := FALSE;   // Q65.0
      "Q65.1" { ExternalVisible := 'False'} : Bool := FALSE;   // Q65.1
      "Q65.2" { ExternalVisible := 'False'} : Bool := FALSE;   // Q65.2
      "Q65.3" { ExternalVisible := 'False'} : Bool := FALSE;   // Q65.3
      "Q65.4" { ExternalVisible := 'False'} : Bool := FALSE;   // Q65.4
      "Q65.5" { ExternalVisible := 'False'} : Bool := FALSE;   // Q65.5
      "Q65.6" { ExternalVisible := 'False'} : Bool := FALSE;   // Q65.6
      "Q65.7" { ExternalVisible := 'False'} : Bool := FALSE;   // Q65.7
      "Q66.0" { ExternalVisible := 'False'} : Bool := FALSE;   // Q66.0
      "Q66.1" { ExternalVisible := 'False'} : Bool := FALSE;   // Q66.1
      "Q66.2" { ExternalVisible := 'False'} : Bool := FALSE;   // Q66.2
      "Q66.3" { ExternalVisible := 'False'} : Bool := FALSE;   // Q66.3
      "Q66.4" { ExternalVisible := 'False'} : Bool := FALSE;   // Q66.4
      "Q66.5" { ExternalVisible := 'False'} : Bool := FALSE;   // Q66.5
      "Q66.6" { ExternalVisible := 'False'} : Bool := FALSE;   // Q66.6
      "Q66.7" { ExternalVisible := 'False'} : Bool := FALSE;   // Q66.7
      "Q67.0" { ExternalVisible := 'False'} : Bool := FALSE;   // Q67.0
      "Q67.1" { ExternalVisible := 'False'} : Bool := FALSE;   // Q67.1
      "Q67.2" { ExternalVisible := 'False'} : Bool := FALSE;   // Q67.2
      "Q67.3" { ExternalVisible := 'False'} : Bool := FALSE;   // Q67.3
      "Q67.4" { ExternalVisible := 'False'} : Bool := FALSE;   // Q67.4
      "Q67.5" { ExternalVisible := 'False'} : Bool := FALSE;   // Q67.5
      "Q67.6" { ExternalVisible := 'False'} : Bool := FALSE;   // Q67.6
      "Q67.7" { ExternalVisible := 'False'} : Bool := FALSE;   // Q67.7
      "Q68.0" { ExternalVisible := 'False'} : Bool := FALSE;   // Q68.0
      "Q68.1" { ExternalVisible := 'False'} : Bool := FALSE;   // Q68.1
      "Q68.2" { ExternalVisible := 'False'} : Bool := FALSE;   // Q68.2
      "Q68.3" { ExternalVisible := 'False'} : Bool := FALSE;   // Q68.3
      "Q68.4" { ExternalVisible := 'False'} : Bool := FALSE;   // Q68.4
      "Q68.5" { ExternalVisible := 'False'} : Bool := FALSE;   // Q68.5
      "Q68.6" { ExternalVisible := 'False'} : Bool := FALSE;   // Q68.6
      "Q68.7" { ExternalVisible := 'False'} : Bool := FALSE;   // Q68.7
      "Q69.0" { ExternalVisible := 'False'} : Bool := FALSE;   // Q69.0
      "Q69.1" { ExternalVisible := 'False'} : Bool := FALSE;   // Q69.1
      "Q69.2" { ExternalVisible := 'False'} : Bool := FALSE;   // Q69.2
      "Q69.3" { ExternalVisible := 'False'} : Bool := FALSE;   // Q69.3
      "Q69.4" { ExternalVisible := 'False'} : Bool := FALSE;   // Q69.4
      "Q69.5" { ExternalVisible := 'False'} : Bool := FALSE;   // Q69.5
      "Q69.6" { ExternalVisible := 'False'} : Bool := FALSE;   // Q69.6
      "Q69.7" { ExternalVisible := 'False'} : Bool := FALSE;   // Q69.7
      "Q70.0" { ExternalVisible := 'False'} : Bool := FALSE;   // Q70.0
      "Q70.1" { ExternalVisible := 'False'} : Bool := FALSE;   // Q70.1
      "Q70.2" { ExternalVisible := 'False'} : Bool := FALSE;   // Q70.2
      "Q70.3" { ExternalVisible := 'False'} : Bool := FALSE;   // Q70.3
      "Q70.4" { ExternalVisible := 'False'} : Bool := FALSE;   // Q70.4
      "Q70.5" { ExternalVisible := 'False'} : Bool := FALSE;   // Q70.5
      "Q70.6" { ExternalVisible := 'False'} : Bool := FALSE;   // Q70.6
      "Q70.7" { ExternalVisible := 'False'} : Bool := FALSE;   // Q70.7
      "Q71.0" { ExternalVisible := 'False'} : Bool := FALSE;   // Q71.0
      "Q71.1" { ExternalVisible := 'False'} : Bool := FALSE;   // Q71.1
      "Q71.2" { ExternalVisible := 'False'} : Bool := FALSE;   // Q71.2
      "Q71.3" { ExternalVisible := 'False'} : Bool := FALSE;   // Q71.3
      "Q71.4" { ExternalVisible := 'False'} : Bool := FALSE;   // Q71.4
      "Q71.5" { ExternalVisible := 'False'} : Bool := FALSE;   // Q71.5
      "Q71.6" { ExternalVisible := 'False'} : Bool := FALSE;   // Q71.6
      "Q71.7" { ExternalVisible := 'False'} : Bool := FALSE;   // Q71.7
      "Q72.0" { ExternalVisible := 'False'} : Bool := FALSE;   // Q72.0
      "Q72.1" { ExternalVisible := 'False'} : Bool := FALSE;   // Q72.1
      "Q72.2" { ExternalVisible := 'False'} : Bool := FALSE;   // Q72.2
      "Q72.3" { ExternalVisible := 'False'} : Bool := FALSE;   // Q72.3
      "Q72.4" { ExternalVisible := 'False'} : Bool := FALSE;   // Q72.4
      "Q72.5" { ExternalVisible := 'False'} : Bool := FALSE;   // Q72.5
      "Q72.6" { ExternalVisible := 'False'} : Bool := FALSE;   // Q72.6
      "Q72.7" { ExternalVisible := 'False'} : Bool := FALSE;   // Q72.7
      "Q73.0" { ExternalVisible := 'False'} : Bool := FALSE;   // Q73.0
      "Q73.1" { ExternalVisible := 'False'} : Bool := FALSE;   // Q73.1
      "Q73.2" { ExternalVisible := 'False'} : Bool := FALSE;   // Q73.2
      "Q73.3" { ExternalVisible := 'False'} : Bool := FALSE;   // Q73.3
      "Q73.4" { ExternalVisible := 'False'} : Bool := FALSE;   // Q73.4
      "Q73.5" { ExternalVisible := 'False'} : Bool := FALSE;   // Q73.5
      "Q73.6" { ExternalVisible := 'False'} : Bool := FALSE;   // Q73.6
      "Q73.7" { ExternalVisible := 'False'} : Bool := FALSE;   // Q73.7
      "Q74.0" { ExternalVisible := 'False'} : Bool := FALSE;   // Q74.0
      "Q74.1" { ExternalVisible := 'False'} : Bool := FALSE;   // Q74.1
      "Q74.2" { ExternalVisible := 'False'} : Bool := FALSE;   // Q74.2
      "Q74.3" { ExternalVisible := 'False'} : Bool := FALSE;   // Q74.3
      "Q74.4" { ExternalVisible := 'False'} : Bool := FALSE;   // Q74.4
      "Q74.5" { ExternalVisible := 'False'} : Bool := FALSE;   // Q74.5
      "Q74.6" { ExternalVisible := 'False'} : Bool := FALSE;   // Q74.6
      "Q74.7" { ExternalVisible := 'False'} : Bool := FALSE;   // Q74.7
      "Q75.0" { ExternalVisible := 'False'} : Bool := FALSE;   // Q75.0
      "Q75.1" { ExternalVisible := 'False'} : Bool := FALSE;   // Q75.1
      "Q75.2" { ExternalVisible := 'False'} : Bool := FALSE;   // Q75.2
      "Q75.3" { ExternalVisible := 'False'} : Bool := FALSE;   // Q75.3
      "Q75.4" { ExternalVisible := 'False'} : Bool := FALSE;   // Q75.4
      "Q75.5" { ExternalVisible := 'False'} : Bool := FALSE;   // Q75.5
      "Q75.6" { ExternalVisible := 'False'} : Bool := FALSE;   // Q75.6
      "Q75.7" { ExternalVisible := 'False'} : Bool := FALSE;   // Q75.7
      "Q76.0" { ExternalVisible := 'False'} : Bool := FALSE;   // Q76.0
      "Q76.1" { ExternalVisible := 'False'} : Bool := FALSE;   // Q76.1
      "Q76.2" { ExternalVisible := 'False'} : Bool := FALSE;   // Q76.2
      "Q76.3" { ExternalVisible := 'False'} : Bool := FALSE;   // Q76.3
      "Q76.4" { ExternalVisible := 'False'} : Bool := FALSE;   // Q76.4
      "Q76.5" { ExternalVisible := 'False'} : Bool := FALSE;   // Q76.5
      "Q76.6" { ExternalVisible := 'False'} : Bool := FALSE;   // Q76.6
      "Q76.7" { ExternalVisible := 'False'} : Bool := FALSE;   // Q76.7
      "Q77.0" { ExternalVisible := 'False'} : Bool := FALSE;   // Q77.0
      "Q77.1" { ExternalVisible := 'False'} : Bool := FALSE;   // Q77.1
      "Q77.2" { ExternalVisible := 'False'} : Bool := FALSE;   // Q77.2
      "Q77.3" { ExternalVisible := 'False'} : Bool := FALSE;   // Q77.3
      "Q77.4" { ExternalVisible := 'False'} : Bool := FALSE;   // Q77.4
      "Q77.5" { ExternalVisible := 'False'} : Bool := FALSE;   // Q77.5
      "Q77.6" { ExternalVisible := 'False'} : Bool := FALSE;   // Q77.6
      "Q77.7" { ExternalVisible := 'False'} : Bool := FALSE;   // Q77.7
      "Q78.0" { ExternalVisible := 'False'} : Bool := FALSE;   // Q78.0
      "Q78.1" { ExternalVisible := 'False'} : Bool := FALSE;   // Q78.1
      "Q78.2" { ExternalVisible := 'False'} : Bool := FALSE;   // Q78.2
      "Q78.3" { ExternalVisible := 'False'} : Bool := FALSE;   // Q78.3
      "Q78.4" { ExternalVisible := 'False'} : Bool := FALSE;   // Q78.4
      "Q78.5" { ExternalVisible := 'False'} : Bool := FALSE;   // Q78.5
      "Q78.6" { ExternalVisible := 'False'} : Bool := FALSE;   // Q78.6
      "Q78.7" { ExternalVisible := 'False'} : Bool := FALSE;   // Q78.7
      "Q79.0" { ExternalVisible := 'False'} : Bool := FALSE;   // Q79.0
      "Q79.1" { ExternalVisible := 'False'} : Bool := FALSE;   // Q79.1
      "Q79.2" { ExternalVisible := 'False'} : Bool := FALSE;   // Q79.2
      "Q79.3" { ExternalVisible := 'False'} : Bool := FALSE;   // Q79.3
      "Q79.4" { ExternalVisible := 'False'} : Bool := FALSE;   // Q79.4
      "Q79.5" { ExternalVisible := 'False'} : Bool := FALSE;   // Q79.5
      "Q79.6" { ExternalVisible := 'False'} : Bool := FALSE;   // Q79.6
      "Q79.7" { ExternalVisible := 'False'} : Bool := FALSE;   // Q79.7
      "Q80.0" { ExternalVisible := 'False'} : Bool := FALSE;   // Q80.0
      "Q80.1" { ExternalVisible := 'False'} : Bool := FALSE;   // Q80.1
      "Q80.2" { ExternalVisible := 'False'} : Bool := FALSE;   // Q80.2
      "Q80.3" { ExternalVisible := 'False'} : Bool := FALSE;   // Q80.3
      "Q80.4" { ExternalVisible := 'False'} : Bool := FALSE;   // Q80.4
      "Q80.5" { ExternalVisible := 'False'} : Bool := FALSE;   // Q80.5
      "Q80.6" { ExternalVisible := 'False'} : Bool := FALSE;   // Q80.6
      "Q80.7" { ExternalVisible := 'False'} : Bool := FALSE;   // Q80.7
      "Q81.0" { ExternalVisible := 'False'} : Bool := FALSE;   // Q81.0
      "Q81.1" { ExternalVisible := 'False'} : Bool := FALSE;   // Q81.1
      "Q81.2" { ExternalVisible := 'False'} : Bool := FALSE;   // Q81.2
      "Q81.3" { ExternalVisible := 'False'} : Bool := FALSE;   // Q81.3
      "Q81.4" { ExternalVisible := 'False'} : Bool := FALSE;   // Q81.4
      "Q81.5" { ExternalVisible := 'False'} : Bool := FALSE;   // Q81.5
      "Q81.6" { ExternalVisible := 'False'} : Bool := FALSE;   // Q81.6
      "Q81.7" { ExternalVisible := 'False'} : Bool := FALSE;   // Q81.7
      "Q82.0" { ExternalVisible := 'False'} : Bool := FALSE;   // Q82.0
      "Q82.1" { ExternalVisible := 'False'} : Bool := FALSE;   // Q82.1
      "Q82.2" { ExternalVisible := 'False'} : Bool := FALSE;   // Q82.2
      "Q82.3" { ExternalVisible := 'False'} : Bool := FALSE;   // Q82.3
      "Q82.4" { ExternalVisible := 'False'} : Bool := FALSE;   // Q82.4
      "Q82.5" { ExternalVisible := 'False'} : Bool := FALSE;   // Q82.5
      "Q82.6" { ExternalVisible := 'False'} : Bool := FALSE;   // Q82.6
      "Q82.7" { ExternalVisible := 'False'} : Bool := FALSE;   // Q82.7
      "Q83.0" { ExternalVisible := 'False'} : Bool := FALSE;   // Q83.0
      "Q83.1" { ExternalVisible := 'False'} : Bool := FALSE;   // Q83.1
      "Q83.2" { ExternalVisible := 'False'} : Bool := FALSE;   // Q83.2
      "Q83.3" { ExternalVisible := 'False'} : Bool := FALSE;   // Q83.3
      "Q83.4" { ExternalVisible := 'False'} : Bool := FALSE;   // Q83.4
      "Q83.5" { ExternalVisible := 'False'} : Bool := FALSE;   // Q83.5
      "Q83.6" { ExternalVisible := 'False'} : Bool := FALSE;   // Q83.6
      "Q83.7" { ExternalVisible := 'False'} : Bool := FALSE;   // Q83.7
      "Q84.0" { ExternalVisible := 'False'} : Bool := FALSE;   // Q84.0
      "Q84.1" { ExternalVisible := 'False'} : Bool := FALSE;   // Q84.1
      "Q84.2" { ExternalVisible := 'False'} : Bool := FALSE;   // Q84.2
      "Q84.3" { ExternalVisible := 'False'} : Bool := FALSE;   // Q84.3
      "Q84.4" { ExternalVisible := 'False'} : Bool := FALSE;   // Q84.4
      "Q84.5" { ExternalVisible := 'False'} : Bool := FALSE;   // Q84.5
      "Q84.6" { ExternalVisible := 'False'} : Bool := FALSE;   // Q84.6
      "Q84.7" { ExternalVisible := 'False'} : Bool := FALSE;   // Q84.7
      "Q85.0" { ExternalVisible := 'False'} : Bool := FALSE;   // Q85.0
      "Q85.1" { ExternalVisible := 'False'} : Bool := FALSE;   // Q85.1
      "Q85.2" { ExternalVisible := 'False'} : Bool := FALSE;   // Q85.2
      "Q85.3" { ExternalVisible := 'False'} : Bool := FALSE;   // Q85.3
      "Q85.4" { ExternalVisible := 'False'} : Bool := FALSE;   // Q85.4
      "Q85.5" { ExternalVisible := 'False'} : Bool := FALSE;   // Q85.5
      "Q85.6" { ExternalVisible := 'False'} : Bool := FALSE;   // Q85.6
      "Q85.7" { ExternalVisible := 'False'} : Bool := FALSE;   // Q85.7
      "Q86.0" { ExternalVisible := 'False'} : Bool := FALSE;   // Q86.0
      "Q86.1" { ExternalVisible := 'False'} : Bool := FALSE;   // Q86.1
      "Q86.2" { ExternalVisible := 'False'} : Bool := FALSE;   // Q86.2
      "Q86.3" { ExternalVisible := 'False'} : Bool := FALSE;   // Q86.3
      "Q86.4" { ExternalVisible := 'False'} : Bool := FALSE;   // Q86.4
      "Q86.5" { ExternalVisible := 'False'} : Bool := FALSE;   // Q86.5
      "Q86.6" { ExternalVisible := 'False'} : Bool := FALSE;   // Q86.6
      "Q86.7" { ExternalVisible := 'False'} : Bool := FALSE;   // Q86.7
      "Q87.0" { ExternalVisible := 'False'} : Bool := FALSE;   // Q87.0
      "Q87.1" { ExternalVisible := 'False'} : Bool := FALSE;   // Q87.1
      "Q87.2" { ExternalVisible := 'False'} : Bool := FALSE;   // Q87.2
      "Q87.3" { ExternalVisible := 'False'} : Bool := FALSE;   // Q87.3
      "Q87.4" { ExternalVisible := 'False'} : Bool := FALSE;   // Q87.4
      "Q87.5" { ExternalVisible := 'False'} : Bool := FALSE;   // Q87.5
      "Q87.6" { ExternalVisible := 'False'} : Bool := FALSE;   // Q87.6
      "Q87.7" { ExternalVisible := 'False'} : Bool := FALSE;   // Q87.7
      "Q88.0" { ExternalVisible := 'False'} : Bool := FALSE;   // Q88.0
      "Q88.1" { ExternalVisible := 'False'} : Bool := FALSE;   // Q88.1
      "Q88.2" { ExternalVisible := 'False'} : Bool := FALSE;   // Q88.2
      "Q88.3" { ExternalVisible := 'False'} : Bool := FALSE;   // Q88.3
      "Q88.4" { ExternalVisible := 'False'} : Bool := FALSE;   // Q88.4
      "Q88.5" { ExternalVisible := 'False'} : Bool := FALSE;   // Q88.5
      "Q88.6" { ExternalVisible := 'False'} : Bool := FALSE;   // Q88.6
      "Q88.7" { ExternalVisible := 'False'} : Bool := FALSE;   // Q88.7
      "Q89.0" { ExternalVisible := 'False'} : Bool := FALSE;   // Q89.0
      "Q89.1" { ExternalVisible := 'False'} : Bool := FALSE;   // Q89.1
      "Q89.2" { ExternalVisible := 'False'} : Bool := FALSE;   // Q89.2
      "Q89.3" { ExternalVisible := 'False'} : Bool := FALSE;   // Q89.3
      "Q89.4" { ExternalVisible := 'False'} : Bool := FALSE;   // Q89.4
      "Q89.5" { ExternalVisible := 'False'} : Bool := FALSE;   // Q89.5
      "Q89.6" { ExternalVisible := 'False'} : Bool := FALSE;   // Q89.6
      "Q89.7" { ExternalVisible := 'False'} : Bool := FALSE;   // Q89.7
      "Q90.0" { ExternalVisible := 'False'} : Bool := FALSE;   // Q90.0
      "Q90.1" { ExternalVisible := 'False'} : Bool := FALSE;   // Q90.1
      "Q90.2" { ExternalVisible := 'False'} : Bool := FALSE;   // Q90.2
      "Q90.3" { ExternalVisible := 'False'} : Bool := FALSE;   // Q90.3
      "Q90.4" { ExternalVisible := 'False'} : Bool := FALSE;   // Q90.4
      "Q90.5" { ExternalVisible := 'False'} : Bool := FALSE;   // Q90.5
      "Q90.6" { ExternalVisible := 'False'} : Bool := FALSE;   // Q90.6
      "Q90.7" { ExternalVisible := 'False'} : Bool := FALSE;   // Q90.7
      "Q91.0" { ExternalVisible := 'False'} : Bool := FALSE;   // Q91.0
      "Q91.1" { ExternalVisible := 'False'} : Bool := FALSE;   // Q91.1
      "Q91.2" { ExternalVisible := 'False'} : Bool := FALSE;   // Q91.2
      "Q91.3" { ExternalVisible := 'False'} : Bool := FALSE;   // Q91.3
      "Q91.4" { ExternalVisible := 'False'} : Bool := FALSE;   // Q91.4
      "Q91.5" { ExternalVisible := 'False'} : Bool := FALSE;   // Q91.5
      "Q91.6" { ExternalVisible := 'False'} : Bool := FALSE;   // Q91.6
      "Q91.7" { ExternalVisible := 'False'} : Bool := FALSE;   // Q91.7
      "Q92.0" { ExternalVisible := 'False'} : Bool := FALSE;   // Q92.0
      "Q92.1" { ExternalVisible := 'False'} : Bool := FALSE;   // Q92.1
      "Q92.2" { ExternalVisible := 'False'} : Bool := FALSE;   // Q92.2
      "Q92.3" { ExternalVisible := 'False'} : Bool := FALSE;   // Q92.3
      "Q92.4" { ExternalVisible := 'False'} : Bool := FALSE;   // Q92.4
      "Q92.5" { ExternalVisible := 'False'} : Bool := FALSE;   // Q92.5
      "Q92.6" { ExternalVisible := 'False'} : Bool := FALSE;   // Q92.6
      "Q92.7" { ExternalVisible := 'False'} : Bool := FALSE;   // Q92.7
      "Q93.0" { ExternalVisible := 'False'} : Bool := FALSE;   // Q93.0
      "Q93.1" { ExternalVisible := 'False'} : Bool := FALSE;   // Q93.1
      "Q93.2" { ExternalVisible := 'False'} : Bool := FALSE;   // Q93.2
      "Q93.3" { ExternalVisible := 'False'} : Bool := FALSE;   // Q93.3
      "Q93.4" { ExternalVisible := 'False'} : Bool := FALSE;   // Q93.4
      "Q93.5" { ExternalVisible := 'False'} : Bool := FALSE;   // Q93.5
      "Q93.6" { ExternalVisible := 'False'} : Bool := FALSE;   // Q93.6
      "Q93.7" { ExternalVisible := 'False'} : Bool := FALSE;   // Q93.7
      "Q94.0" { ExternalVisible := 'False'} : Bool := FALSE;   // Q94.0
      "Q94.1" { ExternalVisible := 'False'} : Bool := FALSE;   // Q94.1
      "Q94.2" { ExternalVisible := 'False'} : Bool := FALSE;   // Q94.2
      "Q94.3" { ExternalVisible := 'False'} : Bool := FALSE;   // Q94.3
      "Q94.4" { ExternalVisible := 'False'} : Bool := FALSE;   // Q94.4
      "Q94.5" { ExternalVisible := 'False'} : Bool := FALSE;   // Q94.5
      "Q94.6" { ExternalVisible := 'False'} : Bool := FALSE;   // Q94.6
      "Q94.7" { ExternalVisible := 'False'} : Bool := FALSE;   // Q94.7
      "Q95.0" { ExternalVisible := 'False'} : Bool := FALSE;   // Q95.0
      "Q95.1" { ExternalVisible := 'False'} : Bool := FALSE;   // Q95.1
      "Q95.2" { ExternalVisible := 'False'} : Bool := FALSE;   // Q95.2
      "Q95.3" { ExternalVisible := 'False'} : Bool := FALSE;   // Q95.3
      "Q95.4" { ExternalVisible := 'False'} : Bool := FALSE;   // Q95.4
      "Q95.5" { ExternalVisible := 'False'} : Bool := FALSE;   // Q95.5
      "Q95.6" { ExternalVisible := 'False'} : Bool := FALSE;   // Q95.6
      "Q95.7" { ExternalVisible := 'False'} : Bool := FALSE;   // Q95.7
      "Q96.0" { ExternalVisible := 'False'} : Bool := FALSE;   // Q96.0
      "Q96.1" { ExternalVisible := 'False'} : Bool := FALSE;   // Q96.1
      "Q96.2" { ExternalVisible := 'False'} : Bool := FALSE;   // Q96.2
      "Q96.3" { ExternalVisible := 'False'} : Bool := FALSE;   // Q96.3
      "Q96.4" { ExternalVisible := 'False'} : Bool := FALSE;   // Q96.4
      "Q96.5" { ExternalVisible := 'False'} : Bool := FALSE;   // Q96.5
      "Q96.6" { ExternalVisible := 'False'} : Bool := FALSE;   // Q96.6
      "Q96.7" { ExternalVisible := 'False'} : Bool := FALSE;   // Q96.7
      "Q97.0" { ExternalVisible := 'False'} : Bool := FALSE;   // Q97.0
      "Q97.1" { ExternalVisible := 'False'} : Bool := FALSE;   // Q97.1
      "Q97.2" { ExternalVisible := 'False'} : Bool := FALSE;   // Q97.2
      "Q97.3" { ExternalVisible := 'False'} : Bool := FALSE;   // Q97.3
      "Q97.4" { ExternalVisible := 'False'} : Bool := FALSE;   // Q97.4
      "Q97.5" { ExternalVisible := 'False'} : Bool := FALSE;   // Q97.5
      "Q97.6" { ExternalVisible := 'False'} : Bool := FALSE;   // Q97.6
      "Q97.7" { ExternalVisible := 'False'} : Bool := FALSE;   // Q97.7
      "Q98.0" { ExternalVisible := 'False'} : Bool := FALSE;   // Q98.0
      "Q98.1" { ExternalVisible := 'False'} : Bool := FALSE;   // Q98.1
      "Q98.2" { ExternalVisible := 'False'} : Bool := FALSE;   // Q98.2
      "Q98.3" { ExternalVisible := 'False'} : Bool := FALSE;   // Q98.3
      "Q98.4" { ExternalVisible := 'False'} : Bool := FALSE;   // Q98.4
      "Q98.5" { ExternalVisible := 'False'} : Bool := FALSE;   // Q98.5
      "Q98.6" { ExternalVisible := 'False'} : Bool := FALSE;   // Q98.6
      "Q98.7" { ExternalVisible := 'False'} : Bool := FALSE;   // Q98.7
      "Q99.0" { ExternalVisible := 'False'} : Bool := FALSE;   // Q99.0
      "Q99.1" { ExternalVisible := 'False'} : Bool := FALSE;   // Q99.1
      "Q99.2" { ExternalVisible := 'False'} : Bool := FALSE;   // Q99.2
      "Q99.3" { ExternalVisible := 'False'} : Bool := FALSE;   // Q99.3
      "Q99.4" { ExternalVisible := 'False'} : Bool := FALSE;   // Q99.4
      "Q99.5" { ExternalVisible := 'False'} : Bool := FALSE;   // Q99.5
      "Q99.6" { ExternalVisible := 'False'} : Bool := FALSE;   // Q99.6
      "Q99.7" { ExternalVisible := 'False'} : Bool := FALSE;   // Q99.7
      "Q100.0" { ExternalVisible := 'False'} : Bool := FALSE;   // Q100.0
      "Q100.1" { ExternalVisible := 'False'} : Bool := FALSE;   // Q100.1
      "Q100.2" { ExternalVisible := 'False'} : Bool := FALSE;   // Q100.2
      "Q100.3" { ExternalVisible := 'False'} : Bool := FALSE;   // Q100.3
      "Q100.4" { ExternalVisible := 'False'} : Bool := FALSE;   // Q100.4
      "Q100.5" { ExternalVisible := 'False'} : Bool := FALSE;   // Q100.5
      "Q100.6" { ExternalVisible := 'False'} : Bool := FALSE;   // Q100.6
      "Q100.7" { ExternalVisible := 'False'} : Bool := FALSE;   // Q100.7
      "Q101.0" { ExternalVisible := 'False'} : Bool := FALSE;   // Q101.0
      "Q101.1" { ExternalVisible := 'False'} : Bool := FALSE;   // Q101.1
